// main statemachine of base controller
CASE me.StateMachine.intState OF
    cSTA_PONBusy: 
        THIS^.sta_PONBusy();
    cSTA_PON: 
        THIS^.sta_PON();
	cSTA_OFFBusy: 
        THIS^.sta_OFFBusy();
    cSTA_OFF: 
        THIS^.sta_OFF();
    cSTA_ERROR: 
        THIS^.sta_ERROR();
    cSTA_ERRORQuit: 
        THIS^.sta_ERRORQuit();
	cSTA_EOFFBusy:
		THIS^.sta_EOFFBusy();
	cSTA_EOFF:
		THIS^.sta_EOFF();
    cSTA_SINGLE_ANSWER: 
        THIS^.sta_SINGLE_ANSWER();
END_CASE;
END_METHOD

END_FUNCTION_BLOCK

// POUs/BaseCtrl/I_CtrlBase
INTERFACE I_CtrlBase

PROPERTY CtrlCIf : POINTER TO T_Ctrl_CIf
GET
END_GET
END_PROPERTY

PROPERTY CtrlFB : POINTER TO FB_CtrlBASE
GET
END_GET
END_PROPERTY

END_INTERFACE

// POUs/Utility/Logger/BasLog/FB_BasLog
FUNCTION_BLOCK FB_BasLog
VAR_INPUT
END_VAR
VAR_OUTPUT
END_VAR
VAR
	stBlClientInfo : T_Bl_LibClient;
	stBlBaseStruct : T_Bl_BaseStruc;
	fbQueue : FB_Queue;
END_VAR

(*__________________________________________________________________________________________________
¦	
¦	Vistaprint Schweiz GmbH
¦	CH - 8401 Winterthur
¦
¦	www.vistaprint.ch - info@vistaprint.ch
¦___________________________________________________________________________________________________

Function desription:
Base logger system. The FUB must be called defined globally one time in PLC-program. After that the implemented 
sender and receiver must interact over the public methodes of the FB_BasLog.

History:
Version		Date			Author		Comment
---------------------------------------------------------------------------------------------------
0.00.1		14.07.2014		AVME/KVO	Start history
___________________________________________________________________________________________________*)

METHOD PUBLIC M_ChangeMask : UINT
VAR_INPUT
	In_strClientName: STRING(Queue.cMAX_NAME_LENGTH); // name of the client
	In_udiNewMask: UDINT;		// new filter mask which log type should be logged for this client
END_VAR
VAR
	usiCnt:USINT;
END_VAR
// change of filter mask
IF (stBlClientInfo.usiClientNr>0) THEN
	FOR usiCnt :=0 TO (stBlClientInfo.usiClientNr-1) BY 1 DO
		IF (In_strClientName=stBlClientInfo.stClient[usiCnt].strName) THEN
			stBlClientInfo.stClient[usiCnt].udiMask := In_udiNewMask;
			M_ChangeMask := 0;
			RETURN;
		END_IF
	END_FOR
END_IF
M_ChangeMask := BasLog.cERR_SYSTEM_NOT_FOUND;
END_METHOD

METHOD PROTECTED M_CheckValidLogType : BOOL
VAR_INPUT
	In_udiLogType : UDINT;
END_VAR
VAR
	ii : UINT;
	udiValue : UDINT := 1;
END_VAR
// check all 2er square
FOR ii :=1 TO 32 BY 1 DO
	// if result identic 
	IF (udiValue=In_udiLogType) THEN
		M_CheckValidLogType := TRUE;
		RETURN;
	END_IF
	udiValue := udiValue * 2; // if not ok multiply with 2
END_FOR
M_CheckValidLogType := FALSE;
END_METHOD

METHOD PUBLIC M_ClientInit : BOOL
VAR_INPUT
	In_strClientName: STRING(Queue.cMAX_NAME_LENGTH); // name of the client
	In_udiMask: UDINT;		// filter mask which log typ should be logged for this client
	In_uinNrOfElement: UINT;	// number of elements in queue
	In_p_fbTimeStamp: POINTER TO FB_TimeStamp; 
	In_bolUseLocalTimeStamp : BOOL; // use local time stamp or UTC
END_VAR
VAR_OUTPUT
	Out_pHandle: POINTER TO T_Queue_Info; 	// handle for read
	Out_uinStatus: UINT;	// feedback value 0:ok
END_VAR
VAR
	usiCnt: USINT;
	pQueueHandle : POINTER TO T_Queue_Info;
	pQueueSysHandle : POINTER TO T_Queue_SysInfo;
	uinStatus : UINT;
END_VAR

// client declaration
IF (stBlClientInfo.usiClientNr>0) THEN
	FOR usiCnt :=0 TO (stBlClientInfo.usiClientNr-1) BY 1 DO
		IF (In_strClientName=stBlClientInfo.stClient[usiCnt].strName) THEN
			// name allready exist - return handle
			Out_pHandle :=  ADR(stBlClientInfo.stHandleRow[0].pQueueHandle[usiCnt]);
			Out_uinStatus := 0;
			RETURN;
		END_IF
	END_FOR
END_IF

// entry timestamp FB
IF (In_p_fbTimeStamp=TC3_MEMMAN.NULL) THEN
	IF (stBlClientInfo.p_fbTimeStamp=TC3_MEMMAN.NULL) THEN
		Out_uinStatus := BasLog.cERR_NO_FB_TIME_STAMP_POINTER;
		RETURN;
	END_IF
ELSE
	stBlClientInfo.p_fbTimeStamp := In_p_fbTimeStamp;
END_IF

	
IF (stBlClientInfo.usiClientNr<BasLog.cMAX_CLIENTS) THEN
	// entry info of new client
	stBlClientInfo.stClient[stBlClientInfo.usiClientNr].strName := In_strClientName;
	stBlClientInfo.stClient[stBlClientInfo.usiClientNr].udiMask := In_udiMask;
	stBlClientInfo.stClient[stBlClientInfo.usiClientNr].udiNrOfElements := In_uinNrOfElement;
	stBlClientInfo.stClient[stBlClientInfo.usiClientNr].bolUseLocalTimeStamp := In_bolUseLocalTimeStamp;
		
	// init queue system if place for new client 
	fbQueue.M_Init(In_strQueueName:=In_strClientName,In_uinNrOfElement:=In_uinNrOfElement,In_udiSizeOfElement:=SIZEOF(T_Bl_BaseStruc),
					In_uinMode:=0,Out_pHandle=>pQueueSysHandle,Out_uinStatus=>uinStatus);
					
	// check feedback from init
	IF (uinStatus<>0) THEN
		Out_uinStatus := uinStatus; // error init queue system
	ELSE
		
		// return handle of TC field zero
		Out_pHandle := ADR(stBlClientInfo.stHandleRow[0].pQueueHandle[stBlClientInfo.usiClientNr]);
		
		// increment client count
		stBlClientInfo.usiClientNr := stBlClientInfo.usiClientNr + 1;
		
		// requirement for handles, if not allready done by tasks
		FOR usiCnt :=0 TO Queue.cMAX_NR_OF_TASKS BY 1 DO
			// if requests allready exist 
			IF (stBlClientInfo.stHandleRow[usiCnt].usiRequest<>0) THEN
				// check for handle
				uinStatus := fbQueue.M_GetHandle_TC(In_strQueueName:=In_strClientName,In_bytTaskIndex:=usiCnt, Out_pQueueHandle=>pQueueHandle);
				
				// check feedback from M_GetHandle_TC
				IF (uinStatus=0) AND (pQueueHandle<>TC3_MEMMAN.NULL) THEN
					// if no error entry handle
					stBlClientInfo.stHandleRow[usiCnt].pQueueHandle[stBlClientInfo.usiClientNr-1] := pQueueHandle;
					stBlClientInfo.stHandleRow[0].pQueueHandle[stBlClientInfo.usiClientNr-1] := pQueueHandle;
				ELSE
					Out_uinStatus := uinStatus; // error M_GetHandle_TC
				END_IF
 			END_IF
		END_FOR
	END_IF
					
ELSE
	Out_uinStatus := BasLog.cERR_TOO_MANY_CLIENTS;
	RETURN;
END_IF
END_METHOD

METHOD PUBLIC M_GetHandle : UINT
VAR_INPUT
;
END_VAR
VAR_OUTPUT
	Out_pHandle : POINTER TO T_Bl_LibHandleRow; // handle of log system for write (M_Log)
END_VAR
VAR
	fbGETCURTASKINDEX : GETCURTASKINDEX;
	usiCnt: USINT;
	pQueueHandle : POINTER TO BYTE;
	uinStatus : UINT;
END_VAR
// get handle of log system
fbGETCURTASKINDEX(); // This function block finds the task index of the task which is called from.
IF (stBlClientInfo.usiClientNr=0) THEN
	// set information that for this taskclass information are requested
	stBlClientInfo.stHandleRow[fbGETCURTASKINDEX.index].usiRequest := 1;
	Out_pHandle := ADR(stBlClientInfo.stHandleRow[fbGETCURTASKINDEX.index]);
ELSE
	// get handle for all declared clients
	FOR usiCnt :=0 TO (stBlClientInfo.usiClientNr-1) BY 1 DO
		M_GetHandle := fbQueue.M_GetHandle(In_strQueueName:=stBlClientInfo.stClient[usiCnt].strName,Out_pQueueHandle=>pQueueHandle);
		
		IF (M_GetHandle=0) AND (pQueueHandle<>TC3_MEMMAN.NULL) THEN
			stBlClientInfo.stHandleRow[fbGETCURTASKINDEX.index].usiRequest := 1;
			stBlClientInfo.stHandleRow[fbGETCURTASKINDEX.index].pQueueHandle[usiCnt] := pQueueHandle;
			
			// handle write in TC 0 writer for reading function
			stBlClientInfo.stHandleRow[0].pQueueHandle[usiCnt] := pQueueHandle;
		ELSE
			RETURN;
		END_IF
	END_FOR
	Out_pHandle := ADR(stBlClientInfo.stHandleRow[fbGETCURTASKINDEX.index]);
END_IF
END_METHOD

METHOD PUBLIC M_Log : UINT
VAR_INPUT
	In_pHandle : POINTER TO BYTE;
	In_udiLogType: UDINT; // log type
	In_intCtrlID: INT; // unique controllerID which has created this entry
	In_strText1: STRING(BasLog.cMAX_CHAR_TEXT1);	//information text1
	In_strText2: STRING(BasLog.cMAX_CHAR_TEXT2); // information text2
	In_dinPar1: DINT; // value parameter  1
	In_dinPar2: DINT; // value parameter  2
	In_dinPar3: DINT; // value parameter  3
	In_dinPar4: DINT; // value parameter  4
END_VAR
VAR
	stTimeStruct: TIMESTRUCT;
	pHandleRow: POINTER TO T_Bl_LibHandleRow;
	usiCnt:USINT;
	uinStatus:UINT;
END_VAR

// check handle ok
IF (In_pHandle=TC3_MEMMAN.NULL) THEN
	M_Log := BasLog.cERR_NO_HANDLE;
	RETURN;
END_IF

// check for correct logtyp
IF ((In_udiLogType>0) AND (M_CheckValidLogType(In_udiLogType)=TRUE))THEN
	// interprete input as row with handles
	pHandleRow := In_pHandle;
	// if time stamp fb is valid
	IF (stBlClientInfo.p_fbTimeStamp<>TC3_MEMMAN.NULL) THEN
		IF (stBlClientInfo.p_fbTimeStamp^.Out_bolInitOk=TRUE) THEN
			IF (stBlClientInfo.stClient[usiCnt].bolUseLocalTimeStamp=FALSE) THEN
				// write time in struct
				stTimeStruct :=  stBlClientInfo.p_fbTimeStamp^.UTC_TimeStruct;
			ELSE
				// write time in struct
				stTimeStruct := stBlClientInfo.p_fbTimeStamp^.LocalTime_TimeStruct_BaseWin;
			END_IF
		ELSE
			M_Log := BasLog.cERR_NO_FB_TIME_STAMP_INIT_NOT_OK;
			RETURN;
		END_IF
	ELSE
		M_Log := BasLog.cERR_NO_FB_TIME_STAMP_POINTER;
		RETURN;
	END_IF
	
	// write parameter and time in struct
	stBlBaseStruct.uinMs := stTimeStruct.wMilliseconds;
	stTimeStruct.wMilliseconds := 0; // The system time has a resolution of 1ms, while the resolution of DATE_AND_TIME is 1s. The milliseconds from the system time are used in the course of the conversion to determine the direction of rounding for the returned DATE_AND_TIME value. Set the wMilliseconds member of the Windows system time structure to zero to deactivate the rounding.
	stBlBaseStruct.dtDateTimeEntry := SYSTEMTIME_TO_DT(stTimeStruct);
	
	stBlBaseStruct.udiLogType := In_udiLogType;
	stBlBaseStruct.intCtrlID := In_intCtrlID;
	stBlBaseStruct.strText1 := In_strText1;
	stBlBaseStruct.strText2 := In_strText2;
	stBlBaseStruct.dinPar1 := In_dinPar1;
	stBlBaseStruct.dinPar2 := In_dinPar2;
	stBlBaseStruct.dinPar3 := In_dinPar3;
	stBlBaseStruct.dinPar4 := In_dinPar4;
	
	// send write command depending on filter mask
	IF (stBlClientInfo.usiClientNr>0) THEN
		FOR usiCnt :=0 TO (stBlClientInfo.usiClientNr-1) BY 1 DO
			// check filter mask
			IF ((In_udiLogType AND stBlClientInfo.stClient[usiCnt].udiMask)<>0) THEN
				uinStatus := fbQueue.M_Write(In_pQueueHandle:=pHandleRow^.pQueueHandle[usiCnt],In_pData:=ADR(stBlBaseStruct));
				IF (uinStatus<>0) THEN
					M_Log := uinStatus;
				END_IF
			END_IF
		END_FOR
	END_IF
ELSE
	M_Log := BasLog.cERR_INVALID_LOGTYPE;
END_IF
END_METHOD

METHOD PUBLIC M_Read : UINT
VAR_INPUT
	In_pHandle : POINTER TO POINTER TO BYTE; // handle for read
	In_pData: POINTER TO T_Bl_BaseStruc; // Pointer for feedback element
END_VAR
VAR
	pReadHandle : POINTER TO POINTER TO T_Queue_Info;
	usiCnt:USINT;
	uinStatus:UINT;
END_VAR

// check handle ok
IF (In_pHandle=TC3_MEMMAN.NULL) THEN
	M_Read := BasLog.cERR_NO_HANDLE;
	RETURN;
END_IF

IF (In_pHandle^=TC3_MEMMAN.NULL) THEN
	M_Read := BasLog.cERR_NO_WRITE_TASK;
	RETURN;
ELSE
	pReadHandle := In_pHandle;
	
	// readout
	M_Read := fbQueue.M_Read(In_pQueueHandle:= pReadHandle^,In_pData:=In_pData); // return<> -> error
END_IF
END_METHOD

END_FUNCTION_BLOCK

// POUs/Utility/Queue/FB_Queue
FUNCTION_BLOCK FB_Queue
VAR // buffer dynamic and PERSISTENT?????
	// creted with new -> dynamic but not retain....arrBuffer: ARRAY[0..ConstBaseLog.MAX_BUFFER_SIZE] OF BYTE; (* Buffer memory used by FB_MemRingBuffer function block *)
	stQueueLibInfo	: T_Queue_LibInfo;
END_VAR

(*__________________________________________________________________________________________________
¦	
¦	Vistaprint Schweiz GmbH
¦	CH - 8401 Winterthur
¦
¦	www.vistaprint.ch - info@vistaprint.ch
¦___________________________________________________________________________________________________

Function desription:
Queue functionallity for mutli tasking system. The FUB must be called defined globally one time in PLC-program. After that the implemented 
sender and receiver must interact over the public methodes.

Public methodes:

M_Clear: 
	Functionality: - Clear all queue entries
	Input parameter: - Queue handlings pointer In_pQueueHandle
	Methode return:	- Status UINT


History:
Version		Date			Author		Comment
---------------------------------------------------------------------------------------------------
0.00.1		14.07.2014		AVME/KVO	Start history
___________________________________________________________________________________________________*)

METHOD FB_exit : BOOL
VAR_INPUT
	bInCopyCode : BOOL; // if TRUE, the exit method is called for exiting an instance that is copied afterwards (online change).
END_VAR
VAR
	pSysInfo : POINTER TO T_Queue_SysInfo;
	pSysInfoNext : POINTER TO T_Queue_SysInfo;
	jj : USINT;
	usiCnt : USINT;
	pDelPointer : POINTER TO BYTE;
	pDelQueueInfo : POINTER TO T_Queue_Info;
END_VAR
END_METHOD

METHOD PROTECTED M_AllocNewQueue : POINTER TO BYTE

VAR_INPUT
	In_udiSizeOfQueue : UDINT; // Byte size of quee to allocate
END_VAR
// Debug counter
stQueueLibInfo.stSysDebugInfo.uinAllocnewQCalls := stQueueLibInfo.stSysDebugInfo.uinAllocnewQCalls + 1;
M_AllocNewQueue := __NEW(BYTE,In_udiSizeOfQueue);

// check if allocate memory is ok
IF (M_AllocNewQueue=TC3_MEMMAN.NULL) THEN
	stQueueLibInfo.uinFUBInternalError := Queue.cERR_MEM_ALLOC;
	M_AllocNewQueue := TC3_MEMMAN.NULL;
END_IF
END_METHOD

METHOD PROTECTED M_AllocNewQueueInfo : POINTER TO T_Queue_Info
VAR_INPUT
END_VAR
VAR
	pSysInfo : POINTER TO T_Queue_SysInfo;
END_VAR
// Debug counter
stQueueLibInfo.stSysDebugInfo.uinAllocNewQICalls := stQueueLibInfo.stSysDebugInfo.uinAllocNewQICalls + 1;

M_AllocNewQueueInfo := __NEW(T_Queue_Info);

// check if allocate memory is ok
IF (M_AllocNewQueueInfo=TC3_MEMMAN.NULL) THEN
	stQueueLibInfo.uinFUBInternalError := Queue.cERR_MEM_ALLOC;
	M_AllocNewQueueInfo := TC3_MEMMAN.NULL;
END_IF
END_METHOD

METHOD PROTECTED M_AllocNewQueueSystem : POINTER TO T_Queue_SysInfo
VAR_INPUT
END_VAR
VAR
	pSysInfo : POINTER TO T_Queue_SysInfo;
END_VAR
// Debug counter
stQueueLibInfo.stSysDebugInfo.uinAllocNewQSCalls := stQueueLibInfo.stSysDebugInfo.uinAllocNewQSCalls + 1;

M_AllocNewQueueSystem := __NEW(T_Queue_SysInfo);

// check if allocate memory is ok
IF (M_AllocNewQueueSystem=TC3_MEMMAN.NULL) THEN
	stQueueLibInfo.uinFUBInternalError := Queue.cERR_MEM_ALLOC;
	M_AllocNewQueueSystem := TC3_MEMMAN.NULL;
END_IF
END_METHOD

METHOD PROTECTED M_CheckAndAppendQueueSysInfo : POINTER TO T_Queue_SysInfo
VAR_INPUT
	In_strQueue : STRING(Queue.cMAX_NAME_LENGTH);
	In_bolCheckOnly : BOOL; // create not automaticallyy a new system -> feedback only valid if exist
END_VAR
VAR
	pSysInfo : POINTER TO T_Queue_SysInfo;
END_VAR
// methode check if queue system allready exist. If not allocate a new one and return pointer.
// Debug counter
stQueueLibInfo.stSysDebugInfo.uinCheckAndAppendQSCalls := stQueueLibInfo.stSysDebugInfo.uinCheckAndAppendQSCalls + 1;

// exist no queue system?
IF (stQueueLibInfo.pstQueue_SysInfo=TC3_MEMMAN.NULL) THEN
	// no queue system exist -> return
	IF (In_bolCheckOnly=TRUE) THEN
		M_CheckAndAppendQueueSysInfo := TC3_MEMMAN.NULL;
		RETURN;
	END_IF
	
	// allocate new queue system
	stQueueLibInfo.pstQueue_SysInfo := M_AllocNewQueueSystem();
	IF (stQueueLibInfo.pstQueue_SysInfo<>TC3_MEMMAN.NULL) THEN
		pSysInfo := stQueueLibInfo.pstQueue_SysInfo;
		// entry queue name
		pSysInfo^.strQueueName := In_strQueue;
		// add secure element
		pSysInfo^.udiSecure := Queue.cSECURE_CODE;
	
		M_CheckAndAppendQueueSysInfo := pSysInfo;
		RETURN;
	ELSE
		M_CheckAndAppendQueueSysInfo := TC3_MEMMAN.NULL;
		RETURN;
	END_IF
END_IF

IF (stQueueLibInfo.pstQueue_SysInfo<>TC3_MEMMAN.NULL) THEN
	// queue system allready exisit
	pSysInfo := stQueueLibInfo.pstQueue_SysInfo;
	
	WHILE (pSysInfo<>TC3_MEMMAN.NULL) DO
		// check queue name
		IF (pSysInfo^.strQueueName = In_strQueue) THEN
			// name found
			M_CheckAndAppendQueueSysInfo := pSysInfo;
			RETURN;
		END_IF
		
		// is this the last element?
		IF (pSysInfo^.pstNextQueue_SysInfo=TC3_MEMMAN.NULL) THEN
			// no queue system exist -> return
			IF (In_bolCheckOnly) THEN
				M_CheckAndAppendQueueSysInfo := TC3_MEMMAN.NULL;
				RETURN;
			END_IF
			
			// allocate new queue system
			pSysInfo^.pstNextQueue_SysInfo := M_AllocNewQueueSystem();
			
			IF (pSysInfo^.pstNextQueue_SysInfo<>TC3_MEMMAN.NULL) THEN
				// reference to new allocated queue system
				pSysInfo := pSysInfo^.pstNextQueue_SysInfo;
				// entry queue name
				pSysInfo^.strQueueName := In_strQueue;
				// add secure element
				pSysInfo^.udiSecure := Queue.cSECURE_CODE;
			
				M_CheckAndAppendQueueSysInfo := pSysInfo;
				RETURN;
			ELSE
				M_CheckAndAppendQueueSysInfo := TC3_MEMMAN.NULL;
				RETURN;
			END_IF
		END_IF
		
		// reference to next element
		pSysInfo := pSysInfo^.pstNextQueue_SysInfo;
	END_WHILE
END_IF

M_CheckAndAppendQueueSysInfo := TC3_MEMMAN.NULL;
END_METHOD

METHOD PUBLIC M_Clear : UINT
VAR_INPUT
	In_pQueueHandle : POINTER TO BYTE; // handle from M_GetHandle()
END_VAR
VAR
	pSysInfo : POINTER TO T_Queue_SysInfo;
	pInfo : POINTER TO T_Queue_Info;
	usiCnt: USINT;
END_VAR
// Clear specific queue system

// check handle ok
IF (In_pQueueHandle=TC3_MEMMAN.NULL) THEN
	M_Clear := Queue.cERR_HANDLE_INVALID;
	RETURN;
END_IF

// handle is pointer to queue info system
pInfo := In_pQueueHandle;

// for reading needed access to system info (check all task class queues)
IF (pInfo^.pQueueSysInfo=TC3_MEMMAN.NULL) THEN
	M_Clear := Queue.cERR_HANDLE_INVALID;
	RETURN;
END_IF

// access system info struct
pSysInfo := pInfo^.pQueueSysInfo;

// validate pointer
IF (pSysInfo^.udiSecure<>Queue.cSECURE_CODE) THEN
	M_Clear := Queue.cERR_HANDLE_INVALID;
	RETURN;
END_IF


// check all queues for first entry
// loop over all queues
FOR usiCnt :=0 TO Queue.cMAX_NR_OF_TASKS BY 1 DO
	pInfo := pSysInfo^.pQueueInfo[usiCnt];
	IF (pInfo<>TC3_MEMMAN.NULL) THEN
		IF (pInfo^.fbBuffer.pBuffer<>TC3_MEMMAN.NULL) THEN
			
			MEMSET( ADR( pInfo^.fbBuffer.pBuffer), 0, pInfo^.fbBuffer.cbBuffer); (* reset (optional) internal buffer *)
			pInfo^.fbBuffer.A_Reset( );
			
			IF (pInfo^.fbBuffer.bOk=TRUE) THEN
				pInfo^.udiFillLevel := (pInfo^.fbBuffer.cbSize * 100) / pInfo^.fbBuffer.cbBuffer; // % 0 empty queue
			ELSE
				M_Clear := Queue.cERR_CLEAR;
				RETURN;
			END_IF
		ELSE
			M_Clear := Queue.cERR_QUEUE_DOES_NOT_EXIST;
			RETURN;
		END_IF
	END_IF
END_FOR
END_METHOD

METHOD PUBLIC M_GetHandle : UINT
VAR_INPUT
	In_strQueueName: STRING(Queue.cMAX_NAME_LENGTH); // name of the queue system
END_VAR
VAR_OUTPUT
	Out_pQueueHandle : POINTER TO T_Queue_Info;
END_VAR
VAR
	fbGETCURTASKINDEX : GETCURTASKINDEX;
END_VAR
// get handle of a specific queue identification over name and task index
fbGETCURTASKINDEX(); // This function block finds the task index of the task which is called from.

// get handle based on task index
M_GetHandle := M_GetHandle_TC(In_strQueueName,fbGETCURTASKINDEX.index,Out_pQueueHandle=>Out_pQueueHandle);
END_METHOD

METHOD PUBLIC M_GetHandle_TC : UINT
VAR_INPUT
	In_strQueueName: STRING(Queue.cMAX_NAME_LENGTH); // name of the queue system
	In_bytTaskIndex: BYTE; // calling task index
END_VAR
VAR_Output
	Out_pQueueHandle : POINTER TO T_Queue_Info;
END_VAR
VAR
	pSysInfo : POINTER TO T_Queue_SysInfo;
	pInfo : POINTER TO T_Queue_Info;
	udiSizeOfQueue: UDINT;
END_VAR
// get handle of a specific queue identification over name and task index

// Debug counter
stQueueLibInfo.stSysDebugInfo.uinGetHandleCalls := stQueueLibInfo.stSysDebugInfo.uinGetHandleCalls + 1;

IF (In_strQueueName='') THEN
	M_GetHandle_TC := Queue.cERR_QUEUE_NAME;
	RETURN;
END_IF
IF (LEN(In_strQueueName)=0) THEN
	M_GetHandle_TC := Queue.cERR_QUEUE_NAME;
	RETURN;
END_IF

// check if queue system allready exist
pSysInfo := M_CheckAndAppendQueueSysInfo(In_strQueueName,FALSE); // false means check if queue system exist!!!

IF (pSysInfo=TC3_MEMMAN.NULL) THEN // system exist?
	M_GetHandle_TC := Queue.cERR_MEM_ALLOC;
	RETURN;
END_IF

// Queue exist and ready?
IF (pSysInfo^.pQueueInfo[In_bytTaskIndex-1]<>TC3_MEMMAN.NULL) THEN
	Out_pQueueHandle := pSysInfo^.pQueueInfo[In_bytTaskIndex-1];
	M_GetHandle_TC := 0;
ELSE
	pSysInfo^.pQueueInfo[In_bytTaskIndex-1] := M_AllocNewQueueInfo();
	
	IF (pSysInfo^.pQueueInfo[In_bytTaskIndex-1] <> TC3_MEMMAN.NULL) THEN
		pInfo := pSysInfo^.pQueueInfo[In_bytTaskIndex-1];
		pInfo^.pQueueSysInfo := pSysInfo; // save system info as reference in queue (parent)
		Out_pQueueHandle := pSysInfo^.pQueueInfo[In_bytTaskIndex-1];	//set pointer feedback
		
		// check if init/size definition allready done
		udiSizeOfQueue := UINT_TO_UDINT(pSysInfo^.uinNbrOfElement)*pSysInfo^.udiSizeOfElement;
		IF (udiSizeOfQueue<>0) THEN
			// Create queue and put reference to info structure
			pInfo^.fbBuffer.pBuffer := M_AllocNewQueue(udiSizeOfQueue);
			IF (pInfo^.fbBuffer.pBuffer<>TC3_MEMMAN.NULL) THEN
				//valid buffer allocated
				pInfo^.fbBuffer.cbBuffer := udiSizeOfQueue; // size created in byte
			ELSE
				M_GetHandle_TC := Queue.cERR_MEM_ALLOC;
				RETURN;
			END_IF
		ELSE
			pInfo^.bolAllocMe := TRUE; // get handle called before valid init done!
		END_IF
	ELSE
		M_GetHandle_TC := Queue.cERR_MEM_ALLOC;
		RETURN;
	END_IF
END_IF
END_METHOD

METHOD PUBLIC M_Init : BOOL
VAR_INPUT
	In_strQueueName: STRING(Queue.cMAX_NAME_LENGTH); // name of the queue system
	In_uinNrOfElement: UINT;		// number of queue element
	In_udiSizeOfElement: UDINT;	// size of an element
	In_uinMode:UINT;				// 0: no overwrite of buffer, 1: ring buffer overwrite oldest entry
END_VAR
VAR_OUTPUT
	Out_pHandle: POINTER TO T_Queue_SysInfo; 			// handle for every task class sender/receiver
	Out_uinStatus: UINT;			// error -> 0:ok
END_VAR
VAR
	pSysInfo : POINTER TO T_Queue_SysInfo;
	pInfo : POINTER TO T_Queue_Info;
	usiCnt: USINT;
	pByte : POINTER TO BYTE;
END_VAR
// Debug counter
stQueueLibInfo.stSysDebugInfo.uinIniCalls := stQueueLibInfo.stSysDebugInfo.uinIniCalls + 1;

IF (In_strQueueName='') THEN
	Out_uinStatus := Queue.cERR_QUEUE_NAME;
	RETURN;
END_IF
IF (LEN(In_strQueueName)=0) THEN
	Out_uinStatus := Queue.cERR_QUEUE_NAME;
	RETURN;
END_IF
IF (In_uinNrOfElement=0) THEN
	Out_uinStatus := Queue.cERR_NR_OF_ELEMENTS;
	RETURN;
END_IF
IF (In_udiSizeOfElement=0) THEN
	Out_uinStatus := Queue.cERR_SIZE_OF_ELEMENTS;
	RETURN;
END_IF

// check if queue system allready exist
pSysInfo := M_CheckAndAppendQueueSysInfo(In_strQueueName,FALSE); // false means check and if not exist create new queeue system!!!

IF (pSysInfo=TC3_MEMMAN.NULL) THEN // system exist
	Out_uinStatus := Queue.cERR_MEM_ALLOC;
	RETURN;
END_IF

// save buffer dimension
pSysInfo^.uinNbrOfElement := In_uinNrOfElement;
pSysInfo^.udiSizeOfElement := In_udiSizeOfElement;
pSysInfo^.uinMode := In_uinMode;

FOR usiCnt :=0 TO Queue.cMAX_NR_OF_TASKS BY 1 DO
	pInfo := pSysInfo^.pQueueInfo[usiCnt]; // Queue info allready allocated -> allocate missing queues for the queue info (init after get_handle)
	IF (pInfo<>TC3_MEMMAN.NULL) THEN // Queue Info allready exist?
		// queue allready allocated?
		IF (pInfo^.fbBuffer.pBuffer=TC3_MEMMAN.NULL) AND (pInfo^.bolAllocMe=TRUE) THEN
			// not allready allocated
			// create FIFO System
			pInfo^.fbBuffer.pBuffer := M_AllocNewQueue(UDINT_TO_UINT(In_uinNrOfElement*In_udiSizeOfElement));
			IF (pInfo^.fbBuffer.pBuffer<>TC3_MEMMAN.NULL) THEN
				//valid buffer allocated
				pInfo^.fbBuffer.cbBuffer := UINT_TO_UDINT(In_uinNrOfElement)*In_udiSizeOfElement; // size created in byte
				pInfo^.bolAllocMe := FALSE;	
			END_IF
		END_IF
	END_IF
END_FOR

Out_uinStatus := 0;
Out_pHandle := pSysInfo;
RETURN;
END_METHOD

METHOD PUBLIC M_Read : UINT
VAR_INPUT
	In_pQueueHandle : POINTER TO BYTE; // handle from M_GetHandle()
	In_pData: POINTER TO BYTE; // destination address of the read element
END_VAR
VAR
	pSysInfo : POINTER TO T_Queue_SysInfo;
	pInfo : POINTER TO T_Queue_Info;
	usiCnt: USINT;
END_VAR
// Reset specific queue system

// check handle ok
IF (In_pQueueHandle=TC3_MEMMAN.NULL) THEN
	M_Read := Queue.cERR_HANDLE_INVALID;
	RETURN;
END_IF

// handle is pointer to queue info system
pInfo := In_pQueueHandle;

// for reading needed access to system info (check all task class queues)
IF (pInfo^.pQueueSysInfo=TC3_MEMMAN.NULL) THEN
	M_Read := Queue.cERR_HANDLE_INVALID;
	RETURN;
END_IF

// access system info struct
pSysInfo := pInfo^.pQueueSysInfo;

// validate pointer
IF (pSysInfo^.udiSecure<>Queue.cSECURE_CODE) THEN
	M_Read := Queue.cERR_HANDLE_INVALID;
	RETURN;
END_IF

//check data read pointer
IF (In_pData=TC3_MEMMAN.NULL) THEN
	M_Read := Queue.cERR_DATA_INVALID;
	RETURN;
END_IF

// check all queues for first entry
// loop over all queues
FOR usiCnt :=0 TO Queue.cMAX_NR_OF_TASKS BY 1 DO
	pInfo := pSysInfo^.pQueueInfo[usiCnt];
	IF (pInfo<>TC3_MEMMAN.NULL) THEN
		
		IF (pInfo^.fbBuffer.pBuffer<>TC3_MEMMAN.NULL) THEN
			
			IF (pInfo^.fbBuffer.nCount>0) THEN // entry?
				pInfo^.fbBuffer.A_RemoveHead(pRead:= In_pData, cbRead:= pSysInfo^.udiSizeOfElement);

				pInfo^.udiFillLevel := (pInfo^.fbBuffer.cbSize * 100) / pInfo^.fbBuffer.cbBuffer;;
				M_Read := 0;
				RETURN;
			END_IF
		ELSE
			M_Read := Queue.cERR_QUEUE_DOES_NOT_EXIST;
			RETURN;
		END_IF
	END_IF
END_FOR

// queue empty
M_Read := Queue.cERR_QUEUE_EMPTY;
END_METHOD

METHOD PUBLIC M_ReadReference : UINT
VAR_INPUT
	In_pQueueHandle : POINTER TO BYTE; // handle from M_GetHandle()
END_VAR
VAR_OUTPUT
	Out_pData: POINTER TO BYTE; // read reference
END_VAR
VAR
	pSysInfo : POINTER TO T_Queue_SysInfo;
	pInfo : POINTER TO T_Queue_Info;
	usiCnt: USINT;
END_VAR
// get reference to element from queue 

// check handle ok
IF (In_pQueueHandle=TC3_MEMMAN.NULL) THEN
	M_ReadReference := Queue.cERR_HANDLE_INVALID;
	RETURN;
END_IF

// handle is pointer to queue info system
pInfo := In_pQueueHandle;

// for reading needed access to system info (check all task class queues)
IF (pInfo^.pQueueSysInfo=TC3_MEMMAN.NULL) THEN
	M_ReadReference := Queue.cERR_HANDLE_INVALID;
	RETURN;
END_IF

// access system info struct
pSysInfo := pInfo^.pQueueSysInfo;

// validate pointer
IF (pSysInfo^.udiSecure<>Queue.cSECURE_CODE) THEN
	M_ReadReference := Queue.cERR_HANDLE_INVALID;
	RETURN;
END_IF

// check all queues for first entry
// loop over all queues
FOR usiCnt :=0 TO Queue.cMAX_NR_OF_TASKS BY 1 DO
	pInfo := pSysInfo^.pQueueInfo[usiCnt];
	IF (pInfo<>TC3_MEMMAN.NULL) THEN
		IF (pInfo^.fbBuffer.pBuffer<>TC3_MEMMAN.NULL) THEN
			
			IF (pInfo^.fbBuffer.nCount>0) THEN // entry?
				pInfo^.fbBuffer.A_GetHead( 	pRead:= Out_pData, cbRead:= pSysInfo^.udiSizeOfElement);
				M_ReadReference := 0;
				RETURN;
			END_IF
		ELSE
			M_ReadReference := Queue.cERR_QUEUE_DOES_NOT_EXIST;
			RETURN;
		END_IF
	END_IF
END_FOR

// queue empty
M_ReadReference := Queue.cERR_QUEUE_EMPTY;
END_METHOD

METHOD PUBLIC M_Write : UINT
VAR_INPUT
	In_pQueueHandle : POINTER TO T_Queue_Info; // handle from M_GetHandle()
	In_pData: POINTER TO BYTE;  // source address of the write element
END_VAR
VAR
	pSysInfo : POINTER TO T_Queue_SysInfo;
	pInfo : POINTER TO T_Queue_Info;
	pData : POINTER TO BYTE; // read dummy element for remove oldest...
END_VAR
// Write element to specific queue system

// check handle ok
IF (In_pQueueHandle=TC3_MEMMAN.NULL) THEN
	M_Write := Queue.cERR_HANDLE_INVALID;
	RETURN;
END_IF

// handle is pointer to queue info system
pInfo := In_pQueueHandle;

// for reading needed access to system info (check all task class queues)
IF (pInfo^.pQueueSysInfo=TC3_MEMMAN.NULL) THEN
	M_Write := Queue.cERR_HANDLE_INVALID;
	RETURN;
END_IF

// access system info struct
pSysInfo := pInfo^.pQueueSysInfo;

// validate pointer
IF (pSysInfo^.udiSecure<>Queue.cSECURE_CODE) THEN
	M_Write := Queue.cERR_HANDLE_INVALID;
	RETURN;
END_IF

//check data
IF (In_pData=TC3_MEMMAN.NULL) THEN
	M_Write := Queue.cERR_DATA_INVALID;
	RETURN;
END_IF

// check if queue exist
IF (pInfo^.fbBuffer.pBuffer=TC3_MEMMAN.NULL) THEN
	M_Write := Queue.cERR_QUEUE_DOES_NOT_EXIST;
	RETURN;
END_IF


// check fill level
// feedback of FIFO = false -> overflow .... IF (pInfo^.udiFillLevel<100) AND (pInfo^.fbBuffer.nCount<pSysInfo^.uinNbrOfElement)THEN
pInfo^.fbBuffer.A_AddTail( pWrite:= In_pData,
				cbWrite:= pSysInfo^.udiSizeOfElement); 
(*				pBuffer:= ADR( arrBuffer ),
				cbBuffer:= SIZEOF( arrBuffer ),
				bOk=> Out_bolOk,
				nCount => Out_udiCount*)
IF (pInfo^.fbBuffer.bOk=FALSE) THEN (* overflow ? *)
	IF (pSysInfo^.uinMode=0) THEN //0:FIFO ring buffer overwrite
		IF (pData = TC3_MEMMAN.NULL) THEN // alloc new dummy read element
			pData := __NEW(BYTE,pSysInfo^.udiSizeOfElement);
		END_IF
		IF (pData <> TC3_MEMMAN.NULL) THEN // alloc new dummy read element
			pInfo^.fbBuffer.A_RemoveHead(pRead:= pData, cbRead:= pSysInfo^.udiSizeOfElement); (* remove one oldest entry *)
			__DELETE(pData); // release dummy memory
			
			pInfo^.fbBuffer.A_AddTail();
			pInfo^.udiFillLevel := (pInfo^.fbBuffer.cbSize * 100) / pInfo^.fbBuffer.cbBuffer;
			M_Write :=0; //Done
		ELSE
			M_Write := Queue.cERR_QUEUE_FULL;
		END_IF
		RETURN;
	ELSE
		pInfo^.udiFillLevel := (pInfo^.fbBuffer.cbSize * 100) / pInfo^.fbBuffer.cbBuffer;
		M_Write := Queue.cERR_QUEUE_FULL;
		RETURN;
	END_IF
ELSE
	pInfo^.udiFillLevel := (pInfo^.fbBuffer.cbSize * 100) / pInfo^.fbBuffer.cbBuffer;
	M_Write :=0; //Done
	RETURN;
END_IF
END_METHOD

END_FUNCTION_BLOCK

// POUs/Utility/getStrInstanceName
FUNCTION getStrInstanceName : T_MaxString
VAR_INPUT
	///'C:\TwinCAT\Plc\Project01\Data.txt';
	strPathName: T_MaxString;
END_VAR
VAR
	strDrive: STRING(3);
	strDir: T_MaxString;
	strFileName: T_MaxString;
	strExt: T_MaxString;
	bolSuccess: BOOL;
END_VAR


bolSuccess := F_SplitPathName( sPathName := strPathName,
                                sDrive := strDrive,
                                sDir := strDir,
                                sFileName := strFileName,
                                sExt := strExt );
								
								getStrInstanceName := MID (strExt,TC2_STANDARD.LEN(strExt),2);

END_FUNCTION

// POUs/Utility/DLL (Double Linked List)/FB_DLL
FUNCTION_BLOCK FB_DLL
VAR
	bDoDataWipe: BOOL := FALSE;
	pFirstElement: POINTER TO T_Element;
	pLastElement: POINTER TO T_Element;
	uiNumberOfElements: UINT;
END_VAR

METHOD addElement : POINTER TO T_Element
VAR_INPUT
	In_pData: POINTER TO BYTE;
	In_uliKey: ULINT;
END_VAR
VAR
	pCurrentElement: POINTER TO T_Element;
END_VAR
addElement := TC3_MEMMAN.NULL;

IF (pFirstElement = TC3_MEMMAN.NULL) THEN
	pCurrentElement := __NEW(T_Element);
	pFirstElement := pCurrentElement;
	pLastElement := pCurrentElement;
	pCurrentElement^.pPrevElement := TC3_MEMMAN.NULL;
	pCurrentElement^.pNextElement := TC3_MEMMAN.NULL;
	pCurrentElement^.pData := In_pData;
	pCurrentElement^.uliKey := In_uliKey;
	addElement := pCurrentElement;
ELSE
	pCurrentElement := __NEW(T_Element);
	pCurrentElement^.pPrevElement := pLastElement;
	pCurrentElement^.pNextElement := TC3_MEMMAN.NULL;
	pCurrentElement^.pData := In_pData;
	pCurrentElement^.uliKey := In_uliKey;
	pLastElement^.pNextElement := pCurrentElement;
	pLastElement := pCurrentElement;
	addElement := pCurrentElement;
END_IF

uiNumberOfElements := uiNumberOfElements + 1;
END_METHOD

METHOD deleteAll : POINTER TO T_Element
WHILE (pFirstElement <> TC3_MEMMAN.NULL) DO
	__DELETE(pFirstElement^.pData);
	deleteElement(pFirstElement);
END_WHILE
END_METHOD

METHOD deleteElement : POINTER TO BYTE
VAR_INPUT
	In_pDeleteElement: POINTER TO T_Element;
END_VAR
deleteElement := In_pDeleteElement^.pData;

IF bDoDataWipe THEN
	IF (In_pDeleteElement^.pData <> TC3_MEMMAN.NULL) THEN
		__DELETE(In_pDeleteElement^.pData);
	END_IF
	deleteElement := TC3_MEMMAN.NULL;
END_IF

IF (In_pDeleteElement = pFirstElement AND In_pDeleteElement = pLastElement) THEN
	pFirstElement := TC3_MEMMAN.NULL;
	pLastElement := TC3_MEMMAN.NULL;
ELSIF (In_pDeleteElement = pFirstElement) THEN
	pFirstElement := In_pDeleteElement^.pNextElement;
	In_pDeleteElement^.pNextElement^.pPrevElement := TC3_MEMMAN.NULL;
ELSIF (In_pDeleteElement = pLastElement) THEN
	pLastElement := In_pDeleteElement^.pPrevElement;
	In_pDeleteElement^.pPrevElement^.pNextElement := TC3_MEMMAN.NULL;
ELSE
	In_pDeleteElement^.pPrevElement^.pNextElement := In_pDeleteElement^.pNextElement;
	In_pDeleteElement^.pNextElement^.pPrevElement := In_pDeleteElement^.pPrevElement;
END_IF

__DELETE(In_pDeleteElement);

uiNumberOfElements := uiNumberOfElements - 1;
END_METHOD

METHOD FB_init : BOOL
VAR_INPUT
	/// if TRUE, the retain variables are initialized (warm start / cold start)
	bInitRetains: BOOL;
	/// if TRUE, the instance afterwards gets moved into the copy code (online change)
	bInCopyCode: BOOL;
	/// if TRUE, the stored data object are automatically deleted
	In_bDoDataWipe: BOOL;
END_VAR
pFirstElement := TC3_MEMMAN.NULL;
pLastElement := TC3_MEMMAN.NULL;
uiNumberOfElements := 0;

bDoDataWipe := In_bDoDataWipe;
END_METHOD

METHOD firstElement : POINTER TO T_Element
firstElement := pFirstElement;
END_METHOD

METHOD numberOfElements : UINT
numberOfElements := uiNumberOfElements;
END_METHOD

METHOD searchElement : POINTER TO T_Element
VAR_INPUT
	In_uliKey: ULINT;
END_VAR
VAR
	pCurrentElement: POINTER TO T_Element;
END_VAR
searchElement := TC3_MEMMAN.NULL;
pCurrentElement := pFirstElement;

WHILE (pCurrentElement <> TC3_MEMMAN.NULL) DO
	IF (pCurrentElement^.uliKey = In_uliKey) THEN
		searchElement := pCurrentElement;
		EXIT;
	END_IF
	pCurrentElement := pCurrentElement^.pNextElement;
END_WHILE
END_METHOD

END_FUNCTION_BLOCK

// POUs/Utility/FileFolder/FB_FileCopy
FUNCTION_BLOCK PUBLIC FB_FileCopy
VAR_INPUT
        srcNetId        : T_AmsNetId;   (* TwinCAT network address of the source file *)
        srcFileName     : T_MaxString;  (* source file path and name *)
        destNetId       : T_AmsNetId;   (* TwinCAT network address of the destination file *)
        destFileName    : T_MaxString;          (* destination file path and name *)
        bExecute        : BOOL;         (* rising edge starts fb execution *)
        tAdsTimeOut     : TIME;         (* ads timeout *)
END_VAR
VAR_OUTPUT
        bBusy           :BOOL;
        bError          :BOOL;
        nErrId          :UDINT;
END_VAR
VAR
        fbFileOpen      :FB_FileOpen;
        fbFileClose     :FB_FileClose;
        fbFileRead      :FB_FileRead;
        fbFileWrite     :FB_FileWrite;

        hSrcFile                :UINT   := 0;(* file handle of the source file *)
        hDestFile               :UINT   := 0;(* file handle of the destination file *)

        Step            :DWORD;
        RisingEdge      :R_TRIG;

        buffRead        :ARRAY[1..10000] OF BYTE;(* buffer *)
        cbReadLength    :UDINT:=0;
END_VAR

(*__________________________________________________________________________________________________
¦	
¦	Vistaprint Schweiz GmbH
¦	CH - 8401 Winterthur
¦
¦	www.vistaprint.ch - info@vistaprint.ch
¦___________________________________________________________________________________________________

Function desription:
	Copy functionality 
	!!!!!!direct source copy from example from Beckhoff -> not Vistaprint notation!!!!
		
History:
Version		Date			Author		Comment
---------------------------------------------------------------------------------------------------
0.00.1		14.05.2014		AVME/KVO	Start history
___________________________________________________________________________________________________*)



RisingEdge(CLK:=bExecute);
IF RisingEdge.Q THEN
        IF NOT bBusy THEN
                bBusy := TRUE;
                bError:= FALSE;
                nErrId:=0;
                Step := 1;
                cbReadLength:=0;
                hSrcFile:=0;
                hDestFile:=0;
        END_IF
END_IF


CASE Step OF
        0:(* do nothing *)
        ;

        1:(* open source file *)
        fbFileOpen(  bExecute := FALSE  );
        fbFileOpen(     sNetId := srcNetId,
                sPathName := srcFileName,
                nMode := FOPEN_MODEREAD OR FOPEN_MODEBINARY,
                ePath := PATH_GENERIC,
                tTimeout := tAdsTimeout,
                bExecute := TRUE );
                Step := Step + 1;

        2:
        fbFileOpen( bExecute := FALSE );
        IF ( NOT fbFileOpen.bBusy ) THEN
                IF ( fbFileOpen.bError ) THEN
                        nErrId := fbFileOpen.nErrId;
                        bError := TRUE;
                        Step := 50;
                ELSE
                        hSrcFile := fbFileOpen.hFile;
                        Step := Step + 1;
                END_IF
        END_IF

        3:(* open destination file *)
        fbFileOpen(  bExecute := FALSE  );
        fbFileOpen(     sNetId := destNetId,
                        sPathName := destFileName,
                        nMode := FOPEN_MODEWRITE OR FOPEN_MODEBINARY,
                        ePath := PATH_GENERIC,
                        tTimeout := tAdsTimeout,
                        bExecute := TRUE );
        Step := Step+1;

        4:
        fbFileOpen(  bExecute := FALSE  );
        IF ( NOT fbFileOpen.bBusy ) THEN
                IF ( fbFileOpen.bError ) THEN
                        nErrId := fbFileOpen.nErrId;
                        bError := TRUE;
                        Step := 50;
                ELSE
                        hDestFile := fbFileOpen.hFile;
                        Step := Step + 1;
                END_IF
        END_IF

        5:(*read data from source file*)
        cbReadLength := 0;
        fbFileRead( bExecute:= FALSE );
        fbFileRead(     sNetId:=SrcNetId,
                        hFile:=hSrcFile,
                        pReadBuff:= ADR(buffRead),
                        cbReadLen:= SIZEOF(buffRead),
                        bExecute:=TRUE,
                        tTimeout:=tAdsTimeOut );
        Step := Step + 1;

        6:
        fbFileRead( bExecute:= FALSE );
        IF ( NOT fbFileRead.bBusy ) THEN
                IF ( fbFileRead.bError ) THEN
                        nErrId := fbFileRead.nErrId;
                        bError := TRUE;
                        Step := 50;
                ELSE
                        cbReadLength := fbFileRead.cbRead;
                        Step := Step + 1;
                END_IF
        END_IF

        7:(*write data to destination file*)
        fbFileWrite( bExecute := FALSE );
        fbFileWrite(    sNetId:=DestNetId,
                        hFile:=hDestFile,
                        pWriteBuff:= ADR(buffRead),
                        cbWriteLen:= cbReadLength,
                        bExecute:=TRUE,
                        tTimeout:=tAdsTimeOut );
        Step := Step + 1;

        8:
        fbFileWrite( bExecute := FALSE );
        IF ( NOT fbFileWrite.bBusy ) THEN
                IF ( fbFileWrite.bError ) THEN
                        nErrId := fbFileWrite.nErrId;
                        bError := TRUE;
                        Step := 50;
                ELSE
                        IF fbFileRead.bEOF THEN (*Check if the EOF flag ist set *)
                                Step := 50;(*cleanup: close the destination and source files *)
                        ELSE
                                Step := 5; (* repeat reading *)
                        END_IF
                END_IF
        END_IF

        30:(* close the destination file *)
        fbFileClose( bExecute := FALSE );
        fbFileClose(    sNetId:=destNetId,
                        hFile:=hDestFile,
                        bExecute:=TRUE,
                        tTimeout:=tAdsTimeOut );
        Step := Step + 1;

        31:
        fbFileClose( bExecute := FALSE );
        IF ( NOT fbFileClose.bBusy ) THEN
                IF ( fbFileClose.bError ) THEN
                        nErrId := fbFileClose.nErrId;
                        bError := TRUE;
                END_IF
                Step := 50;
                hDestFile := 0;
        END_IF

        40: (* close source file *)
        fbFileClose( bExecute := FALSE );
        fbFileClose(    sNetId:=srcNetId,
                        hFile:=hSrcFile,
                        bExecute:=TRUE,
                        tTimeout:=tAdsTimeOut );
        Step := Step + 1;

        41:
        fbFileClose( bExecute := FALSE );
        IF ( NOT fbFileClose.bBusy ) THEN
                IF ( fbFileClose.bError ) THEN
                        nErrId := fbFileClose.nErrId;
                        bError := TRUE;
                END_IF
                Step := 50;
                hSrcFile := 0;
        END_IF

        50: (*error or ready => cleanup*)
        IF ( hDestFile <> 0 ) THEN
                Step := 30; (* close the destination file*)
        ELSIF (hSrcFile <> 0 ) THEN
                Step := 40; (* close the source file *)
        ELSE
                Step := 0;      (* ready *)
                bBusy := FALSE;
        END_IF

END_CASE

END_FUNCTION_BLOCK

// POUs/Utility/FileFolder/FB_FileHdl
FUNCTION_BLOCK FB_FileHdl

VAR_OUTPUT
	Out_bolBusy : BOOL; // busy
	Out_bolNewFileCreated : BOOL; // new file created -> set until next job -> possibility to write header
	Out_udiErrId : UDINT; // error id
	Out_strInfo : STRING; //
END_VAR
VAR
	uinStep : UINT;
	uinStep_old : UINT;
	uinSubStep : UINT;
	intCmd : INT;
	bolInitDone : BOOL;
	strNetId : STRING(23);
	strPathName : T_MaxString; 	// Contains the path and filename for the file to be opened. Note: The path can only point to the local computer’s file system! This means that network paths can not be used here!
	strPath : T_MaxString; 	// Contains only the path 
	strFileName : T_MaxString;	// Contains only the filename
	strFileExt : T_MaxString;	// Contains only the ext
	strPathNameArchive : T_MaxString; // string name of last copied archive file
	strTemp : T_MaxString;
	strFileNameTemp : STRING(200);
	strFullFileName : T_MaxString;
	intLenTemp : INT;
	uin_FileHandle : UINT;	//Contains the file handle created for the file when opening has been successful.
	pWriteBuff: POINTER TO BYTE; // Write buffer adress
	udiWriteLen : UDINT; // Write buffer len
	lreCurFileSize : LREAL;
	stNewestFileEntry : ST_FindFileEntry;
	fbFileOpen_1 : FB_FileOpen;
	fbFileClose_1 : FB_FileClose;
	fbFileWrite_1 : FB_FileWrite;
	fbFileDelete_1 : FB_FileDelete;
	fbFileRename_1 : FB_FileRename;
	fbFileCopy_1 : FB_FileCopy;
	fbFolderHdl_1 : FB_FolderHdl;
	lreMaxFileSize : LREAL := 10; //Bytes? maximal allowed filesize for file -> archivate and deleter or create new
	bolNewFileCreated : BOOL;
	bolTimeRead : BOOL;
	strActualTime : T_MaxString;
	fbNT_GetTime : NT_GetTime;
END_VAR
VAR CONSTANT
	// specific steps definitions
	cStep_Start: UINT := 501;
	cStep_StartReadingFilesInFolder: UINT := 502;
	cStep_ReadingFileInFolder: UINT := 504;
	cStep_FileDelete: UINT := 100;
	cStep_FileClose: UINT := 101;
	cStep_FileOpen: UINT := 102;
	cStep_FileWrite: UINT := 103;
	cStep_NewFile: UINT := 104;
	cStep_FileArchive: UINT := 105;
	cStep_Wait4Job: UINT := 500;
	cStep_Error: UINT := 256;
	
	cSubStep_Done: UINT := 0;
	cSubStep_Finished: UINT := 100;
	cSubStep_Error: UINT := 256;
	
	// configuration constants
	usiMode : UINT := 1; // Mode = 0 logfiles with date, =1 logfile with archive and date
	strSufixArchive : T_MaxString := '_Archive_';

	// commandes constants
	cFILE_HDL_CMD_DONE : INT := -1;
	cFILE_HDL_CMD_WRITE : INT := 1;
	cFILE_HDL_CMD_NEW_FILE : INT := 2;
	cFILE_HDL_CMD_REFRESH_FILE_LIST : INT := 3;
	cFILE_HDL_CMD_CLOSE : INT := 4;
	cFILE_HDL_CMD_FILE_DELETE : INT := 5;
END_VAR

(*__________________________________________________________________________________________________
¦	
¦	Vistaprint Schweiz GmbH
¦	CH - 8401 Winterthur
¦
¦	www.vistaprint.ch - info@vistaprint.ch
¦___________________________________________________________________________________________________

Function desription:
	Manage folder with files: 
	Cyclic Actions:
		- todo evtl. in folder hdl... create folder
		- open file ("a+": Opens for reading and appending; the appending operation includes the removal of the EOF marker before new data is written to the file and the EOF marker is restored after writing is complete; creates the file first if it doesn’t exist.
					When a file is opened with the "a" or "a+" access type, all write operations occur at the end of the file. The file pointer can be repositioned using FB_FileSeek, but is always moved back to the end of the file before any write operation is carried out. Thus, existing data cannot be overwritten.)
		- add buffer to file
		- close file
		- delete file
		- archivate file
		- supervision of active file size
		- todo supervision of nr of entries
		
History:
Version		Date			Author		Comment
---------------------------------------------------------------------------------------------------
0.00.1		13.05.2014		AVME/KVO	Start history
___________________________________________________________________________________________________*)

// read out actual TIME
fbNT_GetTime.START := FALSE;
fbNT_GetTime();
fbNT_GetTime.NETID := '';
fbNT_GetTime.START := TRUE;
fbNT_GetTime.TMOUT := T#500MS;
fbNT_GetTime();

fbFolderHdl_1(); // cyclic call for supervision of numbers of file in folder

CASE uinStep OF
	0:	
		Out_strInfo := 'Wait for init ok -> call methode M_INIT()';
		Out_bolBusy := TRUE;
		IF (bolInitDone=TRUE) AND (fbFolderHdl_1.Out_bolInitDone=TRUE) THEN // refresh file list done
			uinStep := cStep_Start;
		END_IF
		
	cStep_Start: 
		Out_strInfo := 'Start';	
		// entry action
		IF (uinStep<>uinStep_old) THEN
			Out_bolBusy := TRUE;
			Out_udiErrId := 0;
			uinStep_old := uinStep;
			fbFolderHdl_1(); // -> set bol busy
		END_IF

		stNewestFileEntry := fbFolderHdl_1.get_NewestFileEntry; // automatic refresh list!!!
		
		IF ((stNewestFileEntry.sFileName<>'') AND (FIND(stNewestFileEntry.sFileName,strFileName)<>0) AND (FIND(stNewestFileEntry.sFileName,strFileExt)<>0)) THEN // not empty -> found entry and contains IN_strFileName -> no change in config
			IF (usiMode = 0) THEN //new file name with Date and time sufix
				(*???intLenTemp := LEN(stNewestFileEntry.sFileName)-FIND(stNewestFileEntry.sFileName,strFileExt)-1;
				strFileName := stNewestFileEntry.sFileName;
				strFileName := MID (strFileName, 1,intLenTemp); // LEFT doesn't work????
				strPathName := THIS^.M_GetPathName(In_bolSufixDateTime:=FALSE,In_strSufixBeforeDateTime:='');	*)
				strPathName := CONCAT(STR1:=strPath,STR2:=stNewestFileEntry.sFileName);
				lreCurFileSize := UINT64_TO_LREAL(stNewestFileEntry.fileSize); // size of existing file
			ELSE
				// new file name stay always the same -> get size
				strPathName := THIS^.M_GetPathName(In_bolSufixDateTime:=FALSE,In_strSufixBeforeDateTime:='');
				stNewestFileEntry := fbFolderHdl_1.M_getFileInfo(IN_strFileNameWithExt:=strPathName);
				lreCurFileSize := UINT64_TO_LREAL(stNewestFileEntry.fileSize); // size of existing file
			END_IF
			uinStep := cStep_Wait4Job;
		ELSE
			// no matching filename found -> create new file	
			IF (usiMode = 0) THEN // new file name with Date and time sufix
				strPathName := THIS^.M_GetPathName(In_bolSufixDateTime:=TRUE,In_strSufixBeforeDateTime:='_');	
			ELSE	// new file name stay the same but actual file archive with Date and time sufix
				
				strPathName := THIS^.M_GetPathName(In_bolSufixDateTime:=FALSE,In_strSufixBeforeDateTime:='');	
			END_IF
			lreCurFileSize := 0;
			uinStep := cStep_NewFile; // create a new file
		END_IF

	cStep_Wait4Job:	
		Out_strInfo := 'Wait for job';
		// entry action
		IF (uinStep<>uinStep_old) THEN
			Out_bolBusy := FALSE;
			uinSubStep := cSubStep_Done;
			uinStep_old := uinStep;
		END_IF
		
		
		IF (intCmd = cFILE_HDL_CMD_FILE_DELETE) THEN
			Out_bolBusy := TRUE;
			Out_bolNewFileCreated := FALSE;
			uinStep := cStep_FileDelete;
		END_IF
		
		IF (intCmd = cFILE_HDL_CMD_NEW_FILE) THEN
			Out_bolNewFileCreated := FALSE;
			Out_bolBusy := TRUE;
			IF ( uin_FileHandle <> 0 ) THEN // old file still open
				uinStep := cStep_FileClose;
			ELSE
				uinStep := cStep_NewFile;
			END_IF
		END_IF

		IF (intCmd = cFILE_HDL_CMD_WRITE) THEN
			Out_bolNewFileCreated := FALSE;
			Out_bolBusy := TRUE;
			IF ((lreCurFileSize + UDINT_TO_LREAL(udiWriteLen)) > lreMaxFileSize) THEN // supervision of filesize
				IF ( uin_FileHandle <> 0 ) THEN // no file open
					uinStep := cStep_FileClose;
				ELSE
					uinStep := cStep_NewFile;
				END_IF
			ELSE
				IF ( uin_FileHandle <> 0 ) THEN // no file open
					uinStep := cStep_FileWrite;
				ELSE
					uinStep := cStep_FileOpen;
				END_IF
			END_IF
		END_IF
		
		IF (intCmd = cFILE_HDL_CMD_CLOSE) THEN
			Out_bolNewFileCreated := FALSE;
			Out_bolBusy := TRUE;
			uinStep := cStep_FileClose;
		END_IF
		
	cStep_FileDelete:
		Out_strInfo := 'Delete file busy';	
		// entry action
		IF (uinStep<>uinStep_old) THEN
			Out_bolBusy := TRUE;
			uinSubStep := cSubStep_Done;
			uinStep_old := uinStep;
		END_IF
		
		THIS^.M_FileDelete(strNetId,strPathName);
		
		IF (uinSubStep = cSubStep_Finished) THEN
			IF (intCmd = cFILE_HDL_CMD_NEW_FILE) OR (intCmd = cFILE_HDL_CMD_WRITE) THEN
				uinStep := cStep_NewFile;
			ELSE
				uinStep := cStep_Wait4Job; 
			END_IF
		ELSIF (uinSubStep = cSubStep_Error) THEN
			intCmd := cFILE_HDL_CMD_DONE;
			uinStep := cStep_Error;
		END_IF
		
	cStep_NewFile:
		Out_strInfo := 'New file busy';
		// entry action
		IF (uinStep<>uinStep_old) THEN
			Out_bolBusy := TRUE;
			uinSubStep := cSubStep_Done;
			uinStep_old := uinStep;
		END_IF	
		
		lreCurFileSize := 0;
		
		IF (usiMode = 0) THEN // new file name with Date and time sufix
			strPathName := THIS^.M_GetPathName(In_bolSufixDateTime:=TRUE,In_strSufixBeforeDateTime:='');	
		ELSE
			// new file name stay the same but actual file archive with Date and time sufix
			strPathName := THIS^.M_GetPathName(In_bolSufixDateTime:=FALSE,In_strSufixBeforeDateTime:='');	
		END_IF
		
		bolNewFileCreated := TRUE;
		
		IF (intCmd = cFILE_HDL_CMD_WRITE) OR (intCmd = cFILE_HDL_CMD_NEW_FILE) THEN
			IF (usiMode = 0) THEN // new file name with Date and time sufix
				uinStep := cStep_FileOpen;
			ELSE
				uinStep := cStep_FileArchive;
			END_IF
		ELSE
			uinStep := cStep_FileOpen;
		END_IF	
	
	cStep_FileOpen:	
		Out_strInfo := 'Open file busy';
		// entry action
		IF (uinStep<>uinStep_old) THEN
			Out_bolBusy := TRUE;
			uinSubStep := cSubStep_Done;
			uinStep_old := uinStep;
		END_IF	

		THIS^.M_FileOpen(strNetId,strPathName);
		
		IF (uinSubStep = cSubStep_Finished) THEN
			IF (bolNewFileCreated) THEN
				Out_bolNewFileCreated := TRUE;
				bolNewFileCreated := FALSE;
			END_IF
			IF (intCmd = cFILE_HDL_CMD_NEW_FILE) OR (intCmd = cFILE_HDL_CMD_WRITE)THEN
				uinStep := cStep_FileWrite; // refresh actual file list
			ELSE
				intCmd := cFILE_HDL_CMD_DONE;
				uinStep := cStep_Wait4Job;
			END_IF
		ELSIF (uinSubStep = cSubStep_Error) THEN
			intCmd := cFILE_HDL_CMD_DONE;
			uinStep := cStep_Error;
		END_IF	
	
	cStep_FileWrite:	
		Out_strInfo := 'Write file busy';
		// entry action
		IF (uinStep<>uinStep_old) THEN
			Out_bolBusy := TRUE;
			uinSubStep := cSubStep_Done;
			uinStep_old := uinStep;
		END_IF	
		
		THIS^.M_FileWrite();
		
		IF (uinSubStep = cSubStep_Finished) THEN
			intCmd := cFILE_HDL_CMD_DONE;
			uinStep := cStep_FileClose;
		ELSIF (uinSubStep = cSubStep_Error) THEN
			intCmd := cFILE_HDL_CMD_DONE;
			uinStep := cStep_Error;
		END_IF
		
	cStep_FileClose:
		Out_strInfo := 'Close file busy';
		// entry action
		IF (uinStep<>uinStep_old) THEN	
			Out_bolBusy := TRUE;
			uinSubStep := cSubStep_Done;
			uinStep_old := uinStep;
		END_IF	
		
		THIS^.M_FileClose();
		
		IF (uinSubStep = cSubStep_Finished) THEN
			IF (intCmd = cFILE_HDL_CMD_NEW_FILE) OR (intCmd = cFILE_HDL_CMD_WRITE) THEN
				uinStep := cStep_NewFile;
			ELSE
				uinStep := cStep_Wait4Job;
			END_IF
			
		ELSIF (uinSubStep = cSubStep_Error) THEN
			intCmd := cFILE_HDL_CMD_DONE;
			uinStep := cStep_Error;
		END_IF	
		
	cStep_FileArchive:	
		// entry action
		Out_strInfo := 'Archive file busy';
		IF (uinStep<>uinStep_old) THEN	
			Out_bolBusy := TRUE;
			uinSubStep := cSubStep_Done;
			uinStep_old := uinStep;
			strPathNameArchive :=  THIS^.M_GetPathName(In_bolSufixDateTime:=TRUE,In_strSufixBeforeDateTime:=strSufixArchive);
		END_IF	

		// copy takes a lot of time!!! THIS^.M_FileCopy(In_strPathNameSrc := strPathName, In_strPathNameDst :=strPathNameArchive);
		THIS^.M_FileRename(In_strNetId := strNetId,In_strPathNewName:=strPathNameArchive,In_strPathOldName:=strPathName);
		
		IF (uinSubStep = cSubStep_Finished) THEN
			uinStep :=  cStep_FileOpen; // open "new file"// after copy delete original file cStep_FileDelete;
		ELSIF (uinSubStep = cSubStep_Error) THEN
			intCmd := cFILE_HDL_CMD_DONE;
			uinStep := cStep_Error;
		END_IF	
	
	cStep_Error:	
		// entry action
		IF (uinStep<>uinStep_old) THEN
			Out_strInfo := CONCAT(STR1:='Error - ',STR2:= Out_strInfo);
			Out_bolBusy := FALSE;
			uinStep_old := uinStep;
		END_IF
		
		
		IF (intCmd<>cFILE_HDL_CMD_DONE) THEN
			Out_udiErrId := 0;
			uinSubStep := cSubStep_Done;
			IF ( uin_FileHandle <> 0 ) THEN
				uinStep := cStep_FileClose; (* Close the source file *)
			ELSE
				uinStep := cStep_Wait4Job;
			END_IF
		END_IF	
				
END_CASE

PROPERTY PUBLIC ActFileSize : UDINT
GET
ActFileSize := LREAL_TO_UDINT(lreCurFileSize);
END_GET
END_PROPERTY

METHOD PUBLIC M_Cmd_FileDelete : BOOL
VAR_INPUT

END_VAR
intCmd := cFILE_HDL_CMD_FILE_DELETE;
END_METHOD

METHOD PUBLIC M_Cmd_NewFile : BOOL
VAR_INPUT

END_VAR
pWriteBuff := 0;
udiWriteLen := 0;
intCmd := cFILE_HDL_CMD_NEW_FILE;
END_METHOD

METHOD PUBLIC M_Cmd_WriteBuffer : BOOL
VAR_INPUT
	In_p_bytWriteBuff: POINTER TO BYTE;
	In_udiWriteLen : UDINT;
END_VAR
pWriteBuff := In_p_bytWriteBuff;
udiWriteLen := In_udiWriteLen;
intCmd := cFILE_HDL_CMD_WRITE;
END_METHOD

METHOD PROTECTED M_FileClose : BOOL
VAR_INPUT
	 
END_VAR
VAR
	strMyName : STRING := 'M_FileClose: ';
END_VAR
CASE uinSubStep OF
	cSubStep_Done:	
		Out_strInfo :=  CONCAT(CONCAT(Out_strInfo, strMyName) , 'start');
		
		fbFileClose_1.sNetId := fbFileOpen_1.sNetId;
		fbFileClose_1.hFile := uin_FileHandle;
		fbFileClose_1.tTimeout := T#3S;
		fbFileClose_1(bExecute:= FALSE);
		fbFileClose_1(bExecute:= TRUE);
		
		uinSubStep := 1;
		
	1: 
		Out_strInfo :=  CONCAT(CONCAT(Out_strInfo, strMyName) , 'busy');	

		(* wait until function block not busy *)
		fbFileClose_1( bExecute := FALSE );
		IF NOT fbFileClose_1.bBusy THEN
			uin_FileHandle := 0;
			IF NOT fbFileClose_1.bError THEN
				uinSubStep := cSubStep_Finished;
			ELSE 
				Out_udiErrId := fbFileClose_1.nErrID; // 0x703 	Invalid or unknown file handle., 0x70E 	File was opened with wrong method ( e.g. with 'obsolete' FILEOPEN function block ). 
				uinSubStep := cSubStep_Error;
			END_IF
		END_IF
		
	cSubStep_Finished: 
		// succesfully finished
		
	cSubStep_Error:
		Out_strInfo :=  CONCAT(CONCAT(Out_strInfo, strMyName) , CONCAT('error active - number:' , DWORD_TO_HEXSTR( fbFileClose_1.nErrID, 0, FALSE )));
		Out_udiErrId := fbFileClose_1.nErrID;
END_CASE
END_METHOD

METHOD PROTECTED M_FileCopy : BOOL
VAR_INPUT
	 In_strNetIdSrc : STRING(23);
	 In_strPathNameSrc : T_MaxString;
	 In_strNetIdDst : STRING(23);
	 In_strPathNameDst : T_MaxString;
END_VAR
VAR
	strMyName : STRING := 'M_FileCopy: ';
END_VAR
CASE uinSubStep OF
	cSubStep_Done:	
		Out_strInfo :=  CONCAT(CONCAT(Out_strInfo, strMyName) , 'start');
		
		fbFileCopy_1.srcNetId := In_strNetIdSrc; // only local access
		fbFileCopy_1.destNetId := In_strNetIdDst; // only local access
		fbFileCopy_1.srcFileName := In_strPathNameSrc;
		fbFileCopy_1.destFileName := In_strPathNameDst;
		fbFileCopy_1.tAdsTimeOut := T#3S;
		fbFileCopy_1(bExecute:= FALSE);
		fbFileCopy_1(bExecute:= TRUE);
		
		uinSubStep := 1;
		
	1: 
		Out_strInfo :=  CONCAT(CONCAT(Out_strInfo, strMyName) , 'busy');	

		(* wait until function block not busy *)
		fbFileCopy_1( bExecute := FALSE );
		IF NOT fbFileCopy_1.bBusy THEN
			uin_FileHandle := 0;
			IF NOT fbFileCopy_1.bError THEN
				uinSubStep := cSubStep_Finished;
			ELSE 
				Out_udiErrId := fbFileCopy_1.nErrID; 
				uinSubStep := cSubStep_Error;
			END_IF
		END_IF
		
	cSubStep_Finished: 
		// succesfully finished
		
	cSubStep_Error:
		Out_strInfo :=  CONCAT(CONCAT(Out_strInfo, strMyName) , CONCAT('error active - number:' , DWORD_TO_HEXSTR( fbFileCopy_1.nErrID, 0, FALSE )));
		Out_udiErrId := fbFileCopy_1.nErrID;
END_CASE
END_METHOD

METHOD PROTECTED M_FileDelete : BOOL
VAR_INPUT
	In_strNetId : STRING(23);
	In_strPathName : T_MaxString;  
END_VAR
VAR
	strMyName : STRING := 'M_FileDelete: ';
END_VAR

CASE uinSubStep OF
	cSubStep_Done:	
		Out_strInfo :=  CONCAT(CONCAT(Out_strInfo, strMyName) , 'start');
		
		fbFileDelete_1.sNetId :=In_strNetId;
		fbFileDelete_1.sPathName := In_strPathName;
		fbFileDelete_1.ePath := PATH_GENERIC;
		fbFileDelete_1.tTimeout := T#3S;
		fbFileDelete_1(bExecute:= FALSE);
		fbFileDelete_1(bExecute:= TRUE);
		
		uinSubStep := 1;
		
	1: 
		Out_strInfo :=  CONCAT(CONCAT(Out_strInfo, strMyName) , 'busy');	

		(* wait until function block not busy *)
		fbFileDelete_1( bExecute := FALSE );
		IF NOT fbFileDelete_1.bBusy THEN
			IF NOT fbFileDelete_1.bError THEN
				uinSubStep := cSubStep_Finished;
			ELSE 
				Out_udiErrId := fbFileDelete_1.nErrID;
				uinSubStep := cSubStep_Error;
			END_IF
		END_IF
		
	cSubStep_Finished: 
		// succesfully finished
		
	cSubStep_Error:
		Out_strInfo :=  CONCAT(CONCAT(Out_strInfo, strMyName) , CONCAT('error active - number:' , DWORD_TO_HEXSTR( fbFileDelete_1.nErrID, 0, FALSE )));
		Out_udiErrId := fbFileDelete_1.nErrID;
END_CASE
END_METHOD

METHOD PROTECTED M_FileOpen : BOOL
VAR_INPUT
	In_strNetId : STRING(23);
	In_strPathName : T_MaxString;  
END_VAR
VAR
	strMyName : STRING := 'M_FileOpen: ';
END_VAR
CASE uinSubStep OF
	cSubStep_Done:	
		Out_strInfo :=  CONCAT(CONCAT(Out_strInfo, strMyName) , 'start');
		
		fbFileOpen_1.sNetId := In_strNetId;
		fbFileOpen_1.sPathName := In_strPathName;
		fbFileOpen_1.nMode := FOPEN_MODEAPPEND OR FOPEN_MODEPLUS OR FOPEN_MODEBINARY;      // "a+": Opens for reading and appending; the appending operation includes the removal of the EOF marker before new data is written to the file and the EOF marker is restored after writing is complete; creates the file first if it doesn’t exist.
																					// When a file is opened with the "a" or "a+" access type, all write operations occur at the end of the file. The file pointer can be repositioned using FB_FileSeek, but is always moved back to the end of the file before any write operation is carried out. Thus, existing data cannot be overwritten.                       

		fbFileOpen_1.ePath := PATH_GENERIC;
		fbFileOpen_1.tTimeout := T#3S;
		fbFileOpen_1(bExecute:= FALSE);
		fbFileOpen_1(bExecute:= TRUE);
		
		uinSubStep := 1;
		
	1: 
		Out_strInfo :=  CONCAT(CONCAT(Out_strInfo, strMyName) , 'busy');	

		(* wait until function block not busy *)
		fbFileOpen_1( bExecute := FALSE );
		IF NOT fbFileOpen_1.bBusy THEN
			uin_FileHandle := fbFileOpen_1.hFile;
			IF NOT fbFileOpen_1.bError THEN
				uinSubStep := cSubStep_Finished;
			ELSE 
				Out_udiErrId := fbFileOpen_1.nErrID;
				uinSubStep := cSubStep_Error;
			END_IF
		END_IF
		
	cSubStep_Finished: 
		// succesfully finished
		
	cSubStep_Error:
		Out_strInfo :=  CONCAT(CONCAT(Out_strInfo, strMyName) , CONCAT('error active - number:' , DWORD_TO_HEXSTR( fbFileOpen_1.nErrID, 0, FALSE )));
		Out_udiErrId := fbFileOpen_1.nErrID;
END_CASE
END_METHOD

METHOD PROTECTED M_FileRename : BOOL
VAR_INPUT
	 In_strNetId : STRING(23);
	 In_strPathOldName : T_MaxString;
	 In_strPathNewName : T_MaxString;
END_VAR
VAR
	strMyName : STRING := 'M_FileRename: ';
END_VAR
CASE uinSubStep OF
	cSubStep_Done:	
		Out_strInfo :=  CONCAT(CONCAT(Out_strInfo, strMyName) , 'start');
		
		fbFileRename_1.sNetId := In_strNetId;
		fbFileRename_1.sOldName := In_strPathOldName;
		fbFileRename_1.sNewName := In_strPathNewName;
		fbFileRename_1.ePath := PATH_GENERIC;
		fbFileRename_1.tTimeout := T#3S;
		fbFileRename_1(bExecute:= FALSE);
		fbFileRename_1(bExecute:= TRUE);
		
		uinSubStep := 1;
		
	1: 
		Out_strInfo :=  CONCAT(CONCAT(Out_strInfo, strMyName) , 'busy');	

		(* wait until function block not busy *)
		fbFileRename_1( bExecute := FALSE );
		IF NOT fbFileRename_1.bBusy THEN
			IF NOT fbFileRename_1.bError THEN
				uinSubStep := cSubStep_Finished;
			ELSE 
				Out_udiErrId := fbFileRename_1.nErrID;
				uinSubStep := cSubStep_Error;
			END_IF
		END_IF
		
	cSubStep_Finished: 
		// succesfully finished
		
	cSubStep_Error:
		Out_strInfo :=  CONCAT(CONCAT(Out_strInfo, strMyName) , CONCAT('error active - number:' , DWORD_TO_HEXSTR( fbFileRename_1.nErrID, 0, FALSE )));
		Out_udiErrId := fbFileRename_1.nErrID;
END_CASE
END_METHOD

METHOD PROTECTED M_FileWrite : BOOL
VAR_INPUT
	 
END_VAR
VAR
	strMyName : STRING := 'M_FileClose: ';
END_VAR
CASE uinSubStep OF
	cSubStep_Done:	
		Out_strInfo :=  CONCAT(CONCAT(Out_strInfo, strMyName) , 'start');
		
		fbFileWrite_1.sNetId := fbFileOpen_1.sNetId;
		fbFileWrite_1.hFile := uin_FileHandle; // file handle from file open
		fbFileWrite_1.pWriteBuff := pWriteBuff; // Write buffer adress
		fbFileWrite_1.cbWriteLen := udiWriteLen; // Write buffer len
		fbFileWrite_1.tTimeout := T#3S;
		fbFileWrite_1(bExecute:= FALSE);
		fbFileWrite_1(bExecute:= TRUE);
		
		uinSubStep := 1;
		
	1: 
		Out_strInfo :=  CONCAT(CONCAT(Out_strInfo, strMyName) , 'busy');	

		(* wait until function block not busy *)
		fbFileWrite_1( bExecute := FALSE );
		IF NOT fbFileWrite_1.bBusy THEN
			lreCurFileSize := lreCurFileSize + fbFileWrite_1.cbWrite;
			IF NOT fbFileWrite_1.bError THEN
				uinSubStep := cSubStep_Finished;
			ELSE 
				Out_udiErrId := fbFileWrite_1.nErrID; // 0x703 	Invalid or unknown file handle., 0x70E 	File was opened with wrong method ( e.g. with 'obsolete' FILEOPEN function block ). 
				uinSubStep := cSubStep_Error;
			END_IF
		END_IF
		
	cSubStep_Finished: 
		// succesfully finished
		
	cSubStep_Error:
		Out_strInfo :=  CONCAT(CONCAT(Out_strInfo, strMyName) , CONCAT('error active - number:' , DWORD_TO_HEXSTR( fbFileWrite_1.nErrID, 0, FALSE )));
		Out_udiErrId := fbFileOpen_1.nErrID;
END_CASE
END_METHOD

METHOD PRIVATE M_GetPathName : T_MaxString
VAR_INPUT
	In_strSufixBeforeDateTime : T_MaxString;
	In_bolSufixDateTime : BOOL;
END_VAR
VAR
	strTemp: Tc2_System.T_MaxString;
	strTempDateTime: Tc2_System.T_MaxString;
END_VAR

//strPathName := CONCAT(CONCAT(CONCAT(CONCAT(strPath , '\') , strFileName ), '.' ), strFileExt);


strTemp := strPath; //CONCAT(strPath , '\');
strTemp := CONCAT(strTemp , strFileName);
strTemp := CONCAT(strTemp , In_strSufixBeforeDateTime);
IF (In_bolSufixDateTime = TRUE) THEN
	strTempDateTime := '';
	strTempDateTime := CONCAT(strTempDateTime , WORD_TO_STRING(fbNT_GetTime.TIMESTR.wYear));
	IF (fbNT_GetTime.TIMESTR.wMonth<10) THEN
		strTempDateTime := CONCAT(strTempDateTime , '0');
	END_IF
	strTempDateTime := CONCAT(strTempDateTime , WORD_TO_STRING(fbNT_GetTime.TIMESTR.wMonth));
	IF (fbNT_GetTime.TIMESTR.wDay<10) THEN
		strTempDateTime := CONCAT(strTempDateTime , '0');
	END_IF
	strTempDateTime := CONCAT(strTempDateTime , WORD_TO_STRING(fbNT_GetTime.TIMESTR.wDay));
	strTempDateTime := CONCAT(strTempDateTime , '_');
	IF (fbNT_GetTime.TIMESTR.wHour<10) THEN
		strTempDateTime := CONCAT(strTempDateTime , '0');
	END_IF
	strTempDateTime := CONCAT(strTempDateTime , WORD_TO_STRING(fbNT_GetTime.TIMESTR.wHour));
	IF (fbNT_GetTime.TIMESTR.wMinute<10) THEN
		strTempDateTime := CONCAT(strTempDateTime , '0');
	END_IF
	strTempDateTime := CONCAT(strTempDateTime , WORD_TO_STRING(fbNT_GetTime.TIMESTR.wMinute));
	IF (fbNT_GetTime.TIMESTR.wSecond<10) THEN
		strTempDateTime := CONCAT(strTempDateTime , '0');
	END_IF
	strTempDateTime := CONCAT(strTempDateTime , WORD_TO_STRING(fbNT_GetTime.TIMESTR.wSecond));
	strTemp := CONCAT(strTemp , strTempDateTime);
END_IF
strTemp := CONCAT(strTemp , '.');
M_GetPathName := CONCAT(strTemp , strFileExt);
END_METHOD

METHOD PUBLIC M_Init : BOOL
VAR_INPUT
	In_strNetId: STRING(23); // NetId to write to foreign system drives
	IN_strPath : Tc2_System.T_MaxString; 	// Contains only the path 
	IN_strFileName : Tc2_System.T_MaxString;// Contains only the filename
	IN_strFileExt : Tc2_System.T_MaxString;	// Contains only the ext
	IN_uinMaxNrOfFilesInFolder:UINT; // max number of files in folder
	IN_timFileSupervisionPeriod : TIME;// time periode for checking max file nuimber in folder
	IN_lreMaxFileSize : LREAL;// maximal allowed filesize for file -> archivate and deleter or create new
	
END_VAR
strNetId := In_strNetId;
strPath := IN_strPath;
strFileName := IN_strFileName;
strFileExt := IN_strFileExt;
lreMaxFileSize := IN_lreMaxFileSize; // maximal allowed filesize for file -> archivate and deleter or create new

fbFolderHdl_1.M_INIT(IN_strPath := strPath,IN_strPrefixFileName:=strFileName,IN_strFileExt:=strFileExt,In_strNetId:=strNetId);
fbFolderHdl_1.MaxNrOfFilesInFolder := IN_uinMaxNrOfFilesInFolder;
fbFolderHdl_1.FileSupervisionPeriod := IN_timFileSupervisionPeriod;
bolInitDone := TRUE;
END_METHOD

END_FUNCTION_BLOCK

// POUs/Utility/FileFolder/FB_FolderHdl
FUNCTION_BLOCK FB_FolderHdl

VAR_OUTPUT
	Out_bolBusy : BOOL; // busy
	Out_udiErrId : UDINT; // error id
	Out_strInfo : STRING; //
	Out_bolInitDone: BOOL;
END_VAR
VAR
	uinStep: UINT;
	uinStep_old : UINT;
	uinSubStep : UINT;
	intCmd : INT;
	bolInitDone : BOOL;
	bolFileNrExceedArraySize : BOOL; // more than max possibel managed files found -> delete in cyclic
	// configurations/parameters
	strNetId : STRING(23);
	strPath : T_MaxString; 	// Contains only the path 
	strPathName : T_MaxString; 	// Contains the whole search expresion
	strFilePrefix : T_MaxString;	// Contains only the filename
	strFileExt : T_MaxString;	// Contains only the ext
	strTemp : T_MaxString;
	timFileSupervisionPeriod : TIME;
	uinMaxNrOfFilesInFolder : UINT; // max number of files in folder defined
	
	lreTotalFileSize : LREAL;
	aFileList : ARRAY[1..cFILE_HDL_MAX_NR_OF_FILE_TO_MANAGE]  OF ST_FindFileEntry;
	bolAbort : BOOL;
	intOldestFile : INT := 1; // sort list oldest =1
	udiNrOfFilesInFolder : UDINT;

	fbEnumFindFileList_1 : FB_EnumFindFileList;
	fbFileDelete_1 : FB_FileDelete;
	fTON_1 : TON;
	
END_VAR
VAR CONSTANT
	// specific steps definitions
	cStep_Start: UINT := 501;
	cStep_FileDelete: UINT := 100;
	cStep_Refresh: UINT := 101;
	cStep_Wait4Job: UINT := 500;
	cStep_Error: UINT := 256;
	
	cSubStep_Done: UINT := 0;
	cSubStep_Finished: UINT := 100;
	cSubStep_Error: UINT := 256;
	
	
	// commandes constants
	cFOLDER_HDL_CMD_DONE : INT := -1;
	cFOLDER_HDL_CMD_REFRESH_FILE_LIST : INT := 1;
END_VAR

(*__________________________________________________________________________________________________
¦	
¦	Vistaprint Schweiz GmbH
¦	CH - 8401 Winterthur
¦
¦	www.vistaprint.ch - info@vistaprint.ch
¦___________________________________________________________________________________________________

Function desription:
	Manage folder: 
	- Refresh list of files in specific folder
	- sort list form oldest to newest file
	- cyclic supervision of max number of files in folder
	- triggered supervision of max number of files in folder 
		
History:
Version		Date			Author		Comment
---------------------------------------------------------------------------------------------------
0.00.1		14.05.2014		AVME/KVO	Start history
___________________________________________________________________________________________________*)



CASE uinStep OF
	0:	
		// entry action
		IF (uinStep<>uinStep_old) THEN
			Out_strInfo := 'Wait for init ok -> call methode M_INIT()';
			uinSubStep := cSubStep_Done;
			uinStep_old := uinStep;
		END_IF
		
		IF bolInitDone THEN
			uinStep := cStep_Start;
		END_IF
		
	cStep_Start: 
		// entry action
		IF (uinStep<>uinStep_old) THEN
			Out_strInfo := 'Start';	
			Out_bolBusy := 0;
			Out_udiErrId := 0;
			uinSubStep := cSubStep_Done;
			fTON_1.IN := FALSE;
			fTON_1();
			uinStep_old := uinStep;
		END_IF
		
		intCmd := cFOLDER_HDL_CMD_REFRESH_FILE_LIST;// refresh actual file list first

		uinStep := cStep_Wait4Job;
		
	cStep_Wait4Job:	
		// entry action
		IF (uinStep<>uinStep_old) THEN
			Out_strInfo := 'Wait for job';
			Out_bolBusy := FALSE;
			uinSubStep := cSubStep_Done;
			uinStep_old := uinStep;
		END_IF

		IF (timFileSupervisionPeriod>T#0MS) THEN
			fTON_1.PT := timFileSupervisionPeriod;
			fTON_1.IN := TRUE;
			fTON_1();
		END_IF
		
		IF (intCmd = cFOLDER_HDL_CMD_REFRESH_FILE_LIST) OR (fTON_1.Q=TRUE) THEN
			uinStep := cStep_Refresh; // refresh actual file list
		ELSE
			IF (udiNrOfFilesInFolder>uinMaxNrOfFilesInFolder) AND (uinMaxNrOfFilesInFolder<>0) THEN
				intOldestFile := 1; // first entry
				uinStep := cStep_FileDelete;
			END_IF
		END_IF
		
		

	cStep_Refresh:	
		// entry action
		IF (uinStep<>uinStep_old) THEN
			Out_strInfo := 'Refresh file list busy';
			Out_bolBusy := TRUE;
			fTON_1.IN := FALSE;
			fTON_1();
			uinSubStep := cSubStep_Done;
			uinStep_old := uinStep;
		END_IF

		THIS^.M_RefreshFileList();
		
		IF (uinSubStep = cSubStep_Finished) THEN
			THIS^.M_SortFileList();
			intCmd := cFOLDER_HDL_CMD_DONE;
			Out_bolInitDone := TRUE; // valid file list
			uinStep := cStep_Wait4Job;
		ELSIF (uinSubStep = cSubStep_Error) THEN
			intCmd := cFOLDER_HDL_CMD_DONE;
			uinStep := cStep_Error;
		END_IF	

	cStep_FileDelete:
	// entry action
		IF (uinStep<>uinStep_old) THEN
			Out_strInfo := 'Delete file busy';
			Out_bolBusy := TRUE;
			uinSubStep := cSubStep_Done;
			uinStep_old := uinStep;
		END_IF	
		
		strTemp := strPath;
		strTemp := CONCAT(strTemp , aFileList[intOldestFile].sFileName);
		THIS^.M_FileDelete(strTemp);
		
		IF (uinSubStep = cSubStep_Finished) THEN
			intCmd := cFOLDER_HDL_CMD_DONE;
			uinStep := cStep_Refresh; 
		ELSIF (uinSubStep = cSubStep_Error) THEN
			intCmd := cFOLDER_HDL_CMD_DONE;
			uinStep := cStep_Error;
		END_IF
		
	cStep_Error:	
		// entry action
		IF (uinStep<>uinStep_old) THEN
			// written in sub Out_strInfo := 'Error';
			Out_bolBusy := FALSE;
			uinStep_old := uinStep;
		END_IF
		
		IF (intCmd<>cFOLDER_HDL_CMD_DONE) THEN
			Out_udiErrId := 0;
			uinSubStep := cSubStep_Done;
			uinStep := cStep_Wait4Job;
		END_IF
END_CASE

PROPERTY PUBLIC FileSupervisionPeriod : TIME
GET
FileSupervisionPeriod := timFileSupervisionPeriod;
END_GET
SET
timFileSupervisionPeriod := FileSupervisionPeriod;
END_SET
END_PROPERTY

PROPERTY PUBLIC get_FileList : ARRAY[1..cFILE_HDL_MAX_NR_OF_FILE_TO_MANAGE]  OF ST_FindFileEntry;
GET
uinSubStep := 0;

WHILE (THIS^.M_RefreshFileList()=FALSE) DO
	//wait until read all files in folder
END_WHILE

THIS^.M_SortFileList(); // sort last write date -> oldest at position 1!
END_GET
END_PROPERTY

PROPERTY get_NewestFileEntry : ST_FindFileEntry
GET
uinSubStep := 0;
(* läuft nicvht???
WHILE (THIS^.M_RefrehFileList()=FALSE) DO
	//wait until read all files in folder
END_WHILE

THIS^.M_SortFileList(); // sort last write date -> oldest at position 1!
*)
get_NewestFileEntry := aFileList[udiNrOfFilesInFolder];
END_GET
END_PROPERTY

METHOD PUBLIC M_Cmd_RefreshFileList : BOOL
intCmd := cFOLDER_HDL_CMD_REFRESH_FILE_LIST;
END_METHOD

METHOD PROTECTED M_FileDelete : BOOL
VAR_INPUT
	strPathName : T_MaxString;  
END_VAR
VAR
	strMyName : STRING := 'M_FileDelete: ';
END_VAR

CASE uinSubStep OF
	cSubStep_Done:	
		Out_strInfo :=  CONCAT(CONCAT(Out_strInfo, strMyName) , 'start');
		
		fbFileDelete_1.sNetId := strNetId;
		fbFileDelete_1.sPathName := strPathName;
		fbFileDelete_1.ePath := PATH_GENERIC;
		fbFileDelete_1.tTimeout := T#3S;
		fbFileDelete_1(bExecute:= FALSE);
		fbFileDelete_1(bExecute:= TRUE);
		
		uinSubStep := 1;
		
	1: 
		Out_strInfo :=  CONCAT(CONCAT(Out_strInfo, strMyName) , 'busy');	

		(* wait until function block not busy *)
		fbFileDelete_1( bExecute := FALSE );
		IF NOT fbFileDelete_1.bBusy THEN
			IF NOT fbFileDelete_1.bError THEN
				uinSubStep := cSubStep_Finished;
			ELSE 
				Out_udiErrId := fbFileDelete_1.nErrID;
				uinSubStep := cSubStep_Error;
			END_IF
		END_IF
		
	cSubStep_Finished: 
		// succesfully finished
		
	cSubStep_Error:
		Out_strInfo :=  CONCAT(CONCAT(Out_strInfo, strMyName) , CONCAT('error active - number:' , DWORD_TO_HEXSTR( fbFileDelete_1.nErrID, 0, FALSE )));
		Out_udiErrId := fbFileDelete_1.nErrID;
END_CASE
END_METHOD

METHOD PUBLIC M_FileExist : BOOL
VAR_INPUT
	strPathName : Tc2_System.T_MaxString;
END_VAR
VAR
	fbEnum : FB_EnumFindFileEntry := ( sNetID := '', tTimeout := T#5S, sPathName := strPathName );
	uinState : UINT:=0;
END_VAR
WHILE (uinState<>10) DO
	CASE uinState OF
	0:
		fbEnum.sNetId := strNetId;
		fbEnum.eCmd := eEnumCmd_First; (* enum first entry *)
		uinState := 1;
	
	1: (* enum one entry *)
		fbEnum( bExecute := FALSE );
		fbEnum( bExecute := TRUE );
		uinState := 2;
	
	2: (* wait until function block not busy *)
		fbEnum( bExecute := FALSE );
		IF NOT fbEnum.bBusy THEN
			IF NOT fbEnum.bError THEN
				IF NOT fbEnum.bEOE THEN
					M_FileExist := TRUE;
					EXIT;
				ELSE (* no more entries *)
					M_FileExist := FALSE;
					EXIT;
				END_IF
			ELSE (* log error *)
				M_FileExist := FALSE;
				EXIT;
			END_IF
		END_IF
	END_CASE
END_WHILE
END_METHOD

METHOD M_getFileInfo : ST_FindFileEntry
VAR_INPUT
	IN_strFileNameWithExt : Tc2_System.T_MaxString;// Contains the filename with extension
END_VAR
VAR
	ii : UDINT;
	udiUpperLimit : UDINT;
END_VAR
IF (udiNrOfFilesInFolder<cFILE_HDL_MAX_NR_OF_FILE_TO_MANAGE) THEN
	udiUpperLimit := udiNrOfFilesInFolder;
ELSE
	udiUpperLimit := cFILE_HDL_MAX_NR_OF_FILE_TO_MANAGE;	
END_IF

FOR ii:= 0 TO udiUpperLimit DO
	IF (FIND(aFileList[ii].sFileName,IN_strFileNameWithExt)<>0) THEN
		M_getFileInfo := aFileList[ii];
		EXIT;
	END_IF
END_FOR
END_METHOD

METHOD PUBLIC M_GetFileSize : LREAL
VAR_INPUT
	In_strFileName: T_MaxString;
END_VAR
VAR
	i:UDINT;
END_VAR
IF (udiNrOfFilesInFolder=0) THEN
	WHILE (THIS^.M_RefreshFileList()=FALSE) DO
		//wait until read all files in folder
	END_WHILE
END_IF

M_GetFileSize := 0.0;

FOR i := 1 TO udiNrOfFilesInFolder BY 1 DO
	IF (In_strFileName = aFileList[i].sFileName) THEN
		M_GetFileSize := Tc2_Utilities.UINT64_TO_LREAL(aFileList[i].fileSize);
		EXIT;
	END_IF
END_FOR;
END_METHOD

METHOD PUBLIC M_Init : BOOL
VAR_INPUT
	IN_strPath : Tc2_System.T_MaxString; 	// Contains only the path 
	IN_strPrefixFileName : Tc2_System.T_MaxString;// Contains only the filename
	IN_strFileExt : Tc2_System.T_MaxString;	// Contains only the ext
	In_strNetId: STRING(23); // NetId to write to foreign system drives
END_VAR
VAR
	strTemp: Tc2_System.T_MaxString;
END_VAR
strNetId := In_strNetId;
strPath := IN_strPath;
strFilePrefix := IN_strPrefixFileName;
strFileExt := IN_strFileExt;
strTemp := strPath;//todo check path allready added / CONCAT(strPath , '\');
strTemp := CONCAT(strTemp , strFilePrefix);
IF (strFileExt='') THEN
	strPathName := strTemp;
ELSE
	strTemp := CONCAT(strTemp , '.');
	strPathName := CONCAT(strTemp , strFileExt);
END_IF
uinStep := 0;
bolInitDone := TRUE;
END_METHOD

METHOD PUBLIC M_RefreshFileList : BOOL
VAR
	strMyName : STRING := 'M_RefrehFileList: ';
	strTemp : STRING;
END_VAR
CASE uinSubStep OF
	cSubStep_Done:	
		Out_strInfo :=  CONCAT(CONCAT(Out_strInfo, strMyName) , 'start');
		
		M_RefreshFileList := FALSE;
		udiNrOfFilesInFolder := 0;
		
		// define proberties for searching files in folder
		fbEnumFindFileList_1.sNetId := strNetId;

		strTemp := strPath;//todo check path allready added / CONCAT(strPath , '\');
		strTemp := CONCAT(strTemp , strFilePrefix);
		IF (strFileExt='') THEN
			strTemp := CONCAT(strTemp , '*'); // all data types
		ELSE
			strTemp := CONCAT(strTemp , '*.');
			strTemp := CONCAT(strTemp , strFileExt);
		END_IF

		fbEnumFindFileList_1.sPathName := strTemp; // read all files in the defined folder with the defined extension
        fbEnumFindFileList_1.pFindList := ADR(aFileList);
        fbEnumFindFileList_1.cbFindList := SIZEOF(aFileList);
        fbEnumFindFileList_1.tTimeout := DEFAULT_ADS_TIMEOUT;
		fbEnumFindFileList_1.eCmd := E_EnumCmdType.eEnumCmd_First;	(* enum first entry *)
		uinSubStep := 1;
		
	1: 
		Out_strInfo :=  CONCAT(CONCAT(Out_strInfo, strMyName) , 'Reading files in folder busy');	
		
		(* enum one entry *)
		IF bolAbort THEN
			bolAbort := FALSE;
			fbEnumFindFileList_1.eCmd := E_EnumCmdType.eEnumCmd_Abort;
		END_IF
		
		fbEnumFindFileList_1( bExecute := FALSE );
		fbEnumFindFileList_1( bExecute := TRUE );
		uinSubStep := 2;
		
	2:	
		Out_strInfo := CONCAT(CONCAT(Out_strInfo, strMyName) , 'Reading files in folder busy');	
		
		(* wait until function block not busy *)
		fbEnumFindFileList_1( bExecute := FALSE );
		IF NOT fbEnumFindFileList_1.bBusy THEN
			udiNrOfFilesInFolder := fbEnumFindFileList_1.nFindFiles;
			IF NOT fbEnumFindFileList_1.bError THEN
				IF NOT fbEnumFindFileList_1.bEOE THEN
					bolFileNrExceedArraySize := TRUE;
					(* read more informations -> not meaningful 
					fbEnumFindFileList_1.eCmd := E_EnumCmdType.eEnumCmd_Next; (* enum next entry *)
					uinSubStep := 1;*)
					uinSubStep := cSubStep_Finished; // reduce maximum in cyclic actions...-> delete if > max 
				ELSE (* no more entries *)
					uinSubStep := cSubStep_Finished;
				END_IF
			ELSE (* log error *)
				Out_udiErrId := fbEnumFindFileList_1.nErrID;
				uinSubStep := cSubStep_Error;
			END_IF
		END_IF

	cSubStep_Finished: 
		// succesfully finished
		M_RefreshFileList := TRUE;
	cSubStep_Error:
		Out_strInfo :=  CONCAT(CONCAT(Out_strInfo, strMyName) , CONCAT('error active - number:' , DWORD_TO_HEXSTR( fbEnumFindFileList_1.nErrID, 0, FALSE )));
		Out_udiErrId := fbEnumFindFileList_1.nErrID;
		M_RefreshFileList := TRUE;
END_CASE
END_METHOD

METHOD PUBLIC M_SortFileList : BOOL
VAR_INPUT

END_VAR
VAR
	stTempFile 	: ST_FindFileEntry;
	bolNoChangeDone: BOOL;
	i,j :UDINT;
END_VAR
// BubbleSort
M_SortFileList := FALSE;

IF (udiNrOfFilesInFolder>1) THEN
	lreTotalFileSize := UINT64_TO_LREAL(aFileList[1].fileSize);
	FOR i := 1 TO udiNrOfFilesInFolder BY 1 DO
		bolNoChangeDone := TRUE;
		FOR j := 1 TO (udiNrOfFilesInFolder-i) BY 1 DO
			IF (i=1) THEN// count total filesize
				lreTotalFileSize := lreTotalFileSize + Tc2_Utilities.UINT64_TO_LREAL(aFileList[j+1].fileSize);
			END_IF
			
			IF (FILETIME_TO_DT(aFileList[j].lastWriteTime) > FILETIME_TO_DT(aFileList[j + 1].lastWriteTime)) THEN
				// swap files
				memcpy(ADR(stTempFile), ADR(aFileList[j]),SIZEOF(stTempFile));
				memcpy(ADR(aFileList[j]), ADR(aFileList[j + 1]),SIZEOF(stTempFile));
				memcpy(ADR(aFileList[j + 1]), ADR(stTempFile),SIZEOF(stTempFile));
				bolNoChangeDone := FALSE; // at least one change done
			END_IF
			
		END_FOR; 
		IF (bolNoChangeDone) THEN
			EXIT;
		END_IF
	END_FOR;
END_IF;
M_SortFileList := TRUE;
END_METHOD

PROPERTY MaxNrOfFilesInFolder : UINT
GET
MaxNrOfFilesInFolder := uinMaxNrOfFilesInFolder;
END_GET
SET
// not more files allowed as defined in struct....Sort problem
IF (MaxNrOfFilesInFolder<cFILE_HDL_MAX_NR_OF_FILE_TO_MANAGE) THEN
	uinMaxNrOfFilesInFolder := MaxNrOfFilesInFolder;
ELSE
	uinMaxNrOfFilesInFolder := UDINT_TO_UINT(cFILE_HDL_MAX_NR_OF_FILE_TO_MANAGE-1);	
END_IF
END_SET
END_PROPERTY

END_FUNCTION_BLOCK

// POUs/Utility/Logger/BasLog/FB_BasLogTest_Client
FUNCTION_BLOCK FB_BasLogTest_Client
VAR_INPUT
	In_p_fbBasLog: POINTER TO FB_BasLog; // only one central FB_BasLog instance allowed per PLC!!!
END_VAR
VAR_OUTPUT
END_VAR
VAR
	stData : T_Bl_BaseStruc;
	bolInit : BOOL := FALSE;
	pReadHandle : POINTER TO POINTER TO T_Queue_Info;
	uinInitStatus : UINT;
	uinChangeMaskStatus :UINT;
	uinReadStatus : UINT;
	bolChangeMask : BOOL;
	bolRead : BOOL;
	fbTimeStamp: FB_TimeStamp;
END_VAR

(*__________________________________________________________________________________________________
¦	
¦	Vistaprint Schweiz GmbH
¦	CH - 8401 Winterthur
¦
¦	www.vistaprint.ch - info@vistaprint.ch
¦___________________________________________________________________________________________________

Function desription:
Example and test programm for testing the base log system - read data from base log

History:
Version		Date			Author		Comment
---------------------------------------------------------------------------------------------------
0.00.1		14.07.2014		AVME/KVO	Start history
___________________________________________________________________________________________________*)

// system init onetime after start up
IF (bolInit=FALSE) THEN
	// init timer system
	fbTimeStamp.In_strNetId := ''; // use local system time
	fbTimeStamp.In_t_CycleTimeRefreshTimeZone := T#15M; // cyclic check time zone settings
	//init baselog system, one time should be called per baslog system
	In_p_fbBasLog^.M_ClientInit(In_strClientName:='BaseLog',In_udiMask := 16#FFFFFFFF, In_uinNrOfElement:= 128,In_p_fbTimeStamp:=ADR(fbTimeStamp),In_bolUseLocalTimeStamp:=TRUE,Out_pHandle=>pReadHandle,Out_uinStatus=>uinInitStatus);
	
	bolInit := TRUE;
END_IF

fbTimeStamp(); // cyclic call needed for valid time stamp / synchronisation
	
(* change mak on runtime *)
IF (bolRead = TRUE) THEN
	(* cyclically read out of data*)
	uinReadStatus:= In_p_fbBasLog^.M_Read(In_pHandle:=pReadHandle,In_pData:=ADR(stData)); 
END_IF

(* change mak on runtime *)
IF (bolChangeMask = TRUE) THEN
	uinChangeMaskStatus := In_p_fbBasLog^.M_ChangeMask(In_strClientName:='BaseLog',In_udiNewMask:= 16#0F0F0F0F);
	bolChangeMask := FALSE;
END_IF

END_FUNCTION_BLOCK

// POUs/Utility/Logger/BasLog/FB_BasLogTest_Sender
FUNCTION_BLOCK FB_BasLogTest_Sender
VAR_INPUT
	In_p_fbBasLog: POINTER TO FB_BasLog; // only one central FB_BasLog instance allowed per PLC!!!
END_VAR
VAR_OUTPUT
END_VAR
VAR
	bolInit : BOOL := FALSE;
	pHandle : POINTER TO T_Bl_LibHandleRow;
	uinGetHandleStatus : UINT;
	uinWriteStatus :UINT;
	uinDoWrite : UINT;
	dinPar1 : DINT;
	strText1 : STRING(30):='Controller 1';
	strText2 : STRING(30):='Alarm sub info';
END_VAR

(*__________________________________________________________________________________________________
¦	
¦	Vistaprint Schweiz GmbH
¦	CH - 8401 Winterthur
¦
¦	www.vistaprint.ch - info@vistaprint.ch
¦___________________________________________________________________________________________________

Function desription:
Example and test programm for testing the queue system - write data to base log

History:
Version		Date			Author		Comment
---------------------------------------------------------------------------------------------------
0.00.1		14.07.2014		AVME/KVO	Start history
___________________________________________________________________________________________________*)

// system init onetime after start up
IF (bolInit=FALSE) THEN
	uinGetHandleStatus := In_p_fbBasLog^.M_GetHandle(Out_pHandle=>pHandle);
	
	bolInit := TRUE;
END_IF

// write base log entries
IF (uinDoWrite>0) THEN
	uinDoWrite := uinDoWrite - 1;
	dinPar1 := dinPar1 + 1;
	uinWriteStatus := In_p_fbBasLog^.M_Log(In_pHandle:=pHandle,In_udiLogType:=BasLog.cLOGTYPE_ALARM,In_intCtrlID:=11,In_strText1:=strText1,In_strText2:=strText2,In_dinPar1:=dinPar1,In_dinPar2:=0,In_dinPar3:=0,In_dinPar4:=0) ;
END_IF

END_FUNCTION_BLOCK

// POUs/Utility/Logger/DatLog/FB_DatLog
FUNCTION_BLOCK FB_DatLog
VAR_INPUT
END_VAR
VAR_OUTPUT
END_VAR
VAR
	stDatLogLibInfo : T_DL_LibInfo;
	fbPLC_ReadSymInfo: PLC_ReadSymInfoByNameEx; // only one init allowed on the same time....
END_VAR

(*__________________________________________________________________________________________________
¦	
¦	Vistaprint Schweiz GmbH
¦	CH - 8401 Winterthur
¦
¦	www.vistaprint.ch - info@vistaprint.ch
¦___________________________________________________________________________________________________

Function desription:
Base logger system. The FUB must be called defined globally one time in PLC-program. After that the implemented 
sender and receiver must interact over the public methodes of the FB_BasLog.

History:
Version		Date			Author		Comment
---------------------------------------------------------------------------------------------------
0.00.1		14.07.2014		AVME/KVO	Start history
___________________________________________________________________________________________________*)

METHOD PROTECTED M_AllocMEM : POINTER TO BYTE

VAR_INPUT
	In_SizeOfBuffer : UINT; // Byte size of quee to allocate
END_VAR
// Debug counter
M_AllocMEM := __NEW(BYTE,In_SizeOfBuffer);

// check if allocate memory is ok
IF (M_AllocMEM=TC3_MEMMAN.NULL) THEN
	M_AllocMEM := TC3_MEMMAN.NULL;
ELSE
	Tc2_System.MEMSET(M_AllocMEM,0,In_SizeOfBuffer); // init with zero.
END_IF
END_METHOD

METHOD PRIVATE M_CheckAndAppendDatLogInfo : Pointer TO T_DL_SysInfo
VAR_INPUT
	In_strDatLogName: STRING(DatLog.cMAX_SYS_NAME_LENGTH); // name of the client
END_VAR
VAR
	pstSysInfo: POINTER TO T_DL_SysInfo;
END_VAR
// methode check, if data log allready exists and if not allocate a new system
// -> return reference on new system

// exist at least one data log system
IF (stDatLogLibInfo.pstDatLogSysInfo=TC3_MEMMAN.NULL) THEN
	// create  a new system
	stDatLogLibInfo.pstDatLogSysInfo := M_AllocMEM(SIZEOF(T_DL_SysInfo));

	IF (stDatLogLibInfo.pstDatLogSysInfo=TC3_MEMMAN.NULL) THEN
		M_CheckAndAppendDatLogInfo := TC3_MEMMAN.NULL;
		RETURN;
	END_IF
	
	// data log name entry in info system
	stDatLogLibInfo.pstDatLogSysInfo^.strDatLogName := In_strDatLogName;
	M_CheckAndAppendDatLogInfo := stDatLogLibInfo.pstDatLogSysInfo;
	RETURN;
END_IF

// after this point the system has to exist
IF (stDatLogLibInfo.pstDatLogSysInfo<>TC3_MEMMAN.NULL) THEN
	pstSysInfo := stDatLogLibInfo.pstDatLogSysInfo;
	
	WHILE (pstSysInfo<>TC3_MEMMAN.NULL) DO
		IF (pstSysInfo^.strDatLogName=In_strDatLogName) THEN
			// data log name found -> return handle
			M_CheckAndAppendDatLogInfo := pstSysInfo;
			RETURN;
		END_IF
		
		// last element
		IF (pstSysInfo^.pstNextDatLogSystem=TC3_MEMMAN.NULL) THEN
			// the requested log name does not exist -> allocate a new one
			pstSysInfo^.pstNextDatLogSystem := M_AllocMEM(SIZEOF(T_DL_SysInfo));

			IF (pstSysInfo^.pstNextDatLogSystem<>TC3_MEMMAN.NULL) THEN
				pstSysInfo := pstSysInfo^.pstNextDatLogSystem;
				// data log name entry in info system
				pstSysInfo^.strDatLogName := In_strDatLogName;
				M_CheckAndAppendDatLogInfo := pstSysInfo;
				RETURN;
			ELSE
				M_CheckAndAppendDatLogInfo := TC3_MEMMAN.NULL;
				RETURN;
			END_IF
		ELSE
			// reference next
			pstSysInfo := pstSysInfo^.pstNextDatLogSystem;
		END_IF
	END_WHILE
END_IF
END_METHOD

METHOD PUBLIC M_GetHandle : UINT
VAR_INPUT
	In_strDatLogName: STRING(DatLog.cMAX_SYS_NAME_LENGTH); // name of the client
	In_p_fbBasLog: POINTER TO FB_BasLog; // only one central FB_BasLog instance allowed per PLC!!!
END_VAR
VAR_OUTPUT
	Out_pHandle : POINTER TO BYTE; // handle of log system for write (M_Log)
	Out_udiStatus : UDINT; //0 => successful done, <>0 => error
END_VAR
VAR
	pstSysInfo: POINTER TO T_DL_SysInfo;
	uinGetHandleStatus : UINT;
END_VAR

// check if log system allready exists or not, if not allocate a new one
	pstSysInfo := M_CheckAndAppendDatLogInfo(In_strDatLogName:=In_strDatLogName);
	IF (pstSysInfo=TC3_MEMMAN.NULL) THEN
		Out_udiStatus := DatLog.cERR_MEM_ALLOC;
		RETURN;
	END_IF
	
	// log on base log system
	uinGetHandleStatus := In_p_fbBasLog^.M_GetHandle(Out_pHandle=>pstSysInfo^.pBaseLogHandle);
	
	// check error
	IF (uinGetHandleStatus<>0) THEN
		Out_udiStatus := UINT_TO_UDINT(uinGetHandleStatus);
		RETURN;
	ELSE
		pstSysInfo^.p_fbBasLog := In_p_fbBasLog;
		Out_pHandle := pstSysInfo;
	END_IF
END_METHOD

METHOD PUBLIC M_Init : BOOL
VAR_INPUT
	In_bolExecute : BOOL;
	In_strDatLogName: STRING(DatLog.cMAX_SYS_NAME_LENGTH); // name of the client
	In_a_strDataDefinition: ARRAY[0..DatLog.cMAX_NR_OF_VAR] OF STRING(DatLog.cMAX_VAR_NAME_LEN); // complete VarName: p.e.:MAIN.INIT_TASK.VARINT
	In_uinStartId: UINT;	// Start ident for item index -> cfg file config has to match with this number!
	In_Port : T_AmsPort;	// on plc the first runtime system is the 801, 811 ...
END_VAR
VAR_OUTPUT
	Out_udiStatus: UDINT;		 // 0 => successful done, <>0 => error
	Out_bolDone: BOOL;			// Done
END_VAR
VAR
	pstSysInfo: POINTER TO T_DL_SysInfo;
	pstItem : POINTER TO T_DL_Item;
	ii : UINT;
END_VAR

IF (In_bolExecute=TRUE) THEN
	// check if log system allready exists or not, if not allocate a new one
	pstSysInfo := M_CheckAndAppendDatLogInfo(In_strDatLogName:=In_strDatLogName);
	IF (pstSysInfo=TC3_MEMMAN.NULL) THEN
		Out_udiStatus := DatLog.cERR_MEM_ALLOC;
		RETURN;
	END_IF

	IF (stDatLogLibInfo.stStatemachine.bolExecute_old=FALSE) THEN // reset statemachine
		stDatLogLibInfo.stStatemachine.uinState := 1;
		Out_bolDone := FALSE;
		Out_udiStatus := 0;
		stDatLogLibInfo.stStatemachine.usiInitDone := 0;
	END_IF

CASE stDatLogLibInfo.stStatemachine.uinState OF
	1:
		//check number of elements
		FOR ii :=0 TO DatLog.cMAX_NR_OF_VAR BY 1 DO
			IF (In_a_strDataDefinition[ii]='') THEN
				EXIT;
			END_IF
		END_FOR
		
		pstSysInfo^.uinNbrOfItems := ii;
		pstSysInfo^.uinStartId := In_uinStartId;
		
		// allocate memory for items
		pstSysInfo^.pstItems := M_AllocMEM((pstSysInfo^.uinNbrOfItems*SIZEOF(T_DL_Item)));
		IF (pstSysInfo^.pstItems =TC3_MEMMAN.NULL) THEN
			Out_udiStatus := DatLog.cERR_MEM_ALLOC;
			RETURN;
		END_IF
		pstSysInfo^.uinCntReadItems := 0;
		pstSysInfo^.uinItemOffset := 0;
		stDatLogLibInfo.stStatemachine.uinState := stDatLogLibInfo.stStatemachine.uinState + 1;
		
	2:	
		fbPLC_ReadSymInfo.NETID:=''; // local PLC
		IF (In_Port=0) THEN// access first runtime system
			fbPLC_ReadSymInfo.PORT := 851;
		ELSE
			fbPLC_ReadSymInfo.PORT := In_Port;
		END_IF
		fbPLC_ReadSymInfo.SYMNAME := In_a_strDataDefinition[pstSysInfo^.uinCntReadItems];
		fbPLC_ReadSymInfo.START := FALSE;
		fbPLC_ReadSymInfo();
		fbPLC_ReadSymInfo.START := TRUE;
		fbPLC_ReadSymInfo();
		stDatLogLibInfo.stStatemachine.uinState := stDatLogLibInfo.stStatemachine.uinState + 1;
		
	3:
		fbPLC_ReadSymInfo();
		IF (fbPLC_ReadSymInfo.BUSY=FALSE) THEN
			stDatLogLibInfo.stStatemachine.uinState := stDatLogLibInfo.stStatemachine.uinState + 1;
		END_IF
		
	4:
		pstItem := pstSysInfo^.pstItems;
		IF (fbPLC_ReadSymInfo.ERR=FALSE) THEN
			pstItem[pstSysInfo^.uinCntReadItems].strPvName := In_a_strDataDefinition[pstSysInfo^.uinCntReadItems];
			pstItem[pstSysInfo^.uinCntReadItems].uinItemOffset := pstSysInfo^.uinItemOffset;
			pstItem[pstSysInfo^.uinCntReadItems].SymInfo := fbPLC_ReadSymInfo.SYMINFO;
			pstSysInfo^.uinItemOffset := pstSysInfo^.uinItemOffset + UDINT_TO_UINT(pstItem[pstSysInfo^.uinCntReadItems].SymInfo.byteSize); // offset for next
			
			// check if type ok/allowed
			IF (pstItem[pstSysInfo^.uinCntReadItems].SymInfo.symDataType = 'BOOL') THEN 
				pstItem[pstSysInfo^.uinCntReadItems].udiItemType := DatLog.cVAR_TYPE_BOOL;
			ELSIF (pstItem[pstSysInfo^.uinCntReadItems].SymInfo.symDataType = 'SINT') THEN 
				pstItem[pstSysInfo^.uinCntReadItems].udiItemType := DatLog.cVAR_TYPE_SINT;
			ELSIF (pstItem[pstSysInfo^.uinCntReadItems].SymInfo.symDataType = 'INT') THEN 
				pstItem[pstSysInfo^.uinCntReadItems].udiItemType := DatLog.cVAR_TYPE_INT;
			ELSIF (pstItem[pstSysInfo^.uinCntReadItems].SymInfo.symDataType = 'DINT') THEN 
				pstItem[pstSysInfo^.uinCntReadItems].udiItemType := DatLog.cVAR_TYPE_DINT;
			ELSIF (pstItem[pstSysInfo^.uinCntReadItems].SymInfo.symDataType = 'USINT') THEN 
				pstItem[pstSysInfo^.uinCntReadItems].udiItemType := DatLog.cVAR_TYPE_USINT;
			ELSIF (pstItem[pstSysInfo^.uinCntReadItems].SymInfo.symDataType = 'UINT') THEN 
				pstItem[pstSysInfo^.uinCntReadItems].udiItemType := DatLog.cVAR_TYPE_INT;
			ELSIF (pstItem[pstSysInfo^.uinCntReadItems].SymInfo.symDataType = 'UDINT') THEN 
				pstItem[pstSysInfo^.uinCntReadItems].udiItemType := DatLog.cVAR_TYPE_UDINT;
			ELSIF (pstItem[pstSysInfo^.uinCntReadItems].SymInfo.symDataType = 'REAL') THEN 
				pstItem[pstSysInfo^.uinCntReadItems].udiItemType := DatLog.cVAR_TYPE_REAL;
			ELSIF (FIND(STR1:=pstItem[pstSysInfo^.uinCntReadItems].SymInfo.symDataType,STR2:='STRING')<>0) THEN 
				IF (pstItem[pstSysInfo^.uinCntReadItems].SymInfo.byteSize < BasLog.cMAX_CHAR_TEXT2) THEN
					pstItem[pstSysInfo^.uinCntReadItems].udiItemType := DatLog.cVAR_TYPE_STRING;
				ELSE
					Out_udiStatus := DatLog.cERR_UNSUPPORTED_TYPE_STRING_TOO_LONG;
					RETURN;
				END_IF
			ELSE
				Out_udiStatus := DatLog.cERR_UNSUPPORTED_TYPE;
				RETURN;
			END_IF
		ELSE
			Out_udiStatus := fbPLC_ReadSymInfo.ERRID;
			RETURN;
		END_IF
		
		pstSysInfo^.uinCntReadItems := pstSysInfo^.uinCntReadItems  + 1;
		IF (pstSysInfo^.uinCntReadItems<pstSysInfo^.uinNbrOfItems) THEN // read next value
			stDatLogLibInfo.stStatemachine.uinState := 2;
		ELSE
			stDatLogLibInfo.stStatemachine.uinState := stDatLogLibInfo.stStatemachine.uinState + 1; // all items found
		END_IF
	5:
		Out_bolDone := TRUE;
		Out_udiStatus := 0;
		pstSysInfo^.usiInitOk := 1; 
END_CASE
END_IF
stDatLogLibInfo.stStatemachine.bolExecute_old := In_bolExecute;
END_METHOD

METHOD PUBLIC M_Log : UINT
VAR_INPUT
	In_pHandle : POINTER TO BYTE;// handle of log system for write (M_Log)
	In_a_pData: ARRAY [0..DatLog.cMAX_NR_OF_VAR] OF POINTER TO BYTE;// address of structure elements
END_VAR
VAR_OUTPUT
	Out_udiStatus: UDINT;		// 0 => successful done, <>0 => error
END_VAR
VAR
	pstSysInfo: POINTER TO T_DL_SysInfo;
	pstItem : POINTER TO T_DL_Item;
	pstItemEle : T_DL_Item;
	ii : UINT;
	strText2: STRING(BasLog.cMAX_CHAR_TEXT2); // informationtext2
	dinPar2 : DINT;
	dinId : DINT;
	uinStatus : UINT;
END_VAR
// check handle ok
IF (In_pHandle=TC3_MEMMAN.NULL) THEN
	M_Log := DatLog.cERR_NO_HANDLE;
	RETURN;
END_IF

// check data
IF (In_a_pData[0]=TC3_MEMMAN.NULL) THEN
	M_Log := DatLog.cERR_NO_DATE;
	RETURN;
END_IF

// access data loggger system info
pstSysInfo := In_pHandle;

// check if init ok
IF (pstSysInfo^.usiInitOk=0) THEN
	M_Log := DatLog.cERR_INIT_FAILED;
	RETURN;
END_IF

// check if items
IF (pstSysInfo^.pstItems=TC3_MEMMAN.NULL) OR (pstSysInfo^.uinNbrOfItems<=0) THEN
	M_Log := DatLog.cERR_NO_ITEMS;
	RETURN;
END_IF
// access item definitions
pstItem := pstSysInfo^.pstItems;

// inc. record id: important the id is inc bevor and after writing of data -> to be sure that no second write is done (MUTEX)
stDatLogLibInfo.udiCommonRecIdx := stDatLogLibInfo.udiCommonRecIdx + 1;
IF (stDatLogLibInfo.udiCommonRecIdx=0) THEN
	stDatLogLibInfo.udiCommonRecIdx := stDatLogLibInfo.udiCommonRecIdx + 1;
END_IF
// write record start
// AE_BL_VAR_TYPE_CMD_NEW_REC
uinStatus := pstSysInfo^.p_fbBasLog^.M_Log(In_pHandle := pstSysInfo^.pBaseLogHandle,In_udiLogType:=BasLog.cLOGTYPE_DATA,In_intCtrlID:=DatLog.cCTRL_ID,In_strText1:='DataLog',In_strText2:='AE_BL_VAR_TYPE_CMD_NEW_REC',In_dinPar1:=0,In_dinPar2:=0,In_dinPar3:=BasLog.cVAR_TYPE_CMD_NEW_REC,In_dinPar4:=UDINT_TO_DINT(stDatLogLibInfo.udiCommonRecIdx));
IF (uinStatus<>0) THEN
	M_Log := uinStatus;
	RETURN;
END_IF

// loop over all items and write data to logger
FOR ii :=0 TO (pstSysInfo^.uinNbrOfItems-1) BY 1 DO
	// write item
	pstItemEle := pstItem[ii]; // for debugging
	// id
	dinId := UINT_TO_DINT(pstSysInfo^.uinStartId + ii);
	IF (pstItem[ii].udiItemType=DatLog.cVAR_TYPE_STRING) THEN
		MEMSET(destAddr:=ADR(strText2),fillByte:=0,n:= SIZEOF(strText2)); // to be sure that a zero is at the end
		// doesn't work with beckhoff...MEMCPY(destAddr := ADR(strText2),srcAddr:= (In_pAdrData + pstItem[ii].uinItemOffset),n:=pstItem[ii].SymInfo.byteSize);
		MEMCPY(destAddr := ADR(strText2),srcAddr:= In_a_pData[ii],n:=pstItem[ii].SymInfo.byteSize);
		dinPar2 := 0;
	ELSE
		strText2 := pstItem[ii].strPvName; // just for info
		MEMCPY(destAddr := ADR(dinPar2),srcAddr:= In_a_pData[ii],n:=pstItem[ii].SymInfo.byteSize);
	END_IF
	
	// log item
	uinStatus := pstSysInfo^.p_fbBasLog^.M_Log(In_pHandle := pstSysInfo^.pBaseLogHandle,In_udiLogType:=BasLog.cLOGTYPE_DATA,In_intCtrlID:=DatLog.cCTRL_ID,In_strText1:='DataLog',In_strText2:=strText2,In_dinPar1:=dinId,In_dinPar2:=dinPar2,In_dinPar3:=UDINT_TO_DINT(pstItem[ii].udiItemType),In_dinPar4:=UDINT_TO_DINT(stDatLogLibInfo.udiCommonRecIdx));

	IF (uinStatus<>0) THEN // no stop write error number
		M_Log := uinStatus;
	END_IF
END_FOR

// write record stop
// AE_BL_VAR_TYPE_CMD_NEW_REC
uinStatus := pstSysInfo^.p_fbBasLog^.M_Log(In_pHandle := pstSysInfo^.pBaseLogHandle,In_udiLogType:=BasLog.cLOGTYPE_DATA,In_intCtrlID:=DatLog.cCTRL_ID,In_strText1:='DataLog',In_strText2:='AE_BL_VAR_TYPE_CMD_END_REC',In_dinPar1:=0,In_dinPar2:=0,In_dinPar3:=BasLog.cVAR_TYPE_CMD_END_REC,In_dinPar4:=UDINT_TO_DINT(stDatLogLibInfo.udiCommonRecIdx));
IF (uinStatus<>0) THEN
	M_Log := uinStatus;
	RETURN;
END_IF

// increment id a second time
stDatLogLibInfo.udiCommonRecIdx := stDatLogLibInfo.udiCommonRecIdx + 1;
IF (stDatLogLibInfo.udiCommonRecIdx=0) THEN
	stDatLogLibInfo.udiCommonRecIdx := stDatLogLibInfo.udiCommonRecIdx + 1;
END_IF
END_METHOD

END_FUNCTION_BLOCK

// POUs/Utility/Logger/DatLog/FB_DatLogTest_Sender
FUNCTION_BLOCK FB_DatLogTest_Sender
VAR_INPUT
	In_p_fbBasLog: POINTER TO FB_BasLog; // only one central FB_BasLog instance allowed per PLC!!!
	In_a_pData: ARRAY [0..DatLog.cMAX_NR_OF_VAR] OF POINTER TO BYTE;
	In_strTaskName: STRING(20);
	In_strValueNameOfData: STRING(20);
END_VAR
VAR_OUTPUT
	Out_bolInit : BOOL := FALSE;
END_VAR
VAR
	bolDone : BOOL;
	pDL_Handle: POINTER TO T_DL_SysInfo;
	udiStatusInit :UDINT;
	udiStatus : UDINT;
	fbDatLog: FB_DatLog;
	a_strDataDefinition :ARRAY[0..DatLog.cMAX_NR_OF_VAR] OF STRING(DatLog.cMAX_VAR_NAME_LEN);
	uinDoLogData : UINT;
	strTemp: T_MaxString;
	strTemp2: T_MaxString;
	ii : UINT;
END_VAR

(*__________________________________________________________________________________________________
¦	
¦	Vistaprint Schweiz GmbH
¦	CH - 8401 Winterthur
¦
¦	www.vistaprint.ch - info@vistaprint.ch
¦___________________________________________________________________________________________________

Function desription:
Example and test programm for testing the data logger system - write data to data log

History:
Version		Date			Author		Comment
---------------------------------------------------------------------------------------------------
0.00.1		02.09.2014		AVME/KVO	Start history
___________________________________________________________________________________________________*)

// system init onetime after start up
IF (Out_bolInit=FALSE) THEN
	
	// TODO :parse a struct on PLC...
	FOR ii := 0 TO DatLog.cMAX_NR_OF_VAR DO
		strTemp := In_strTaskName;
		strTemp := CONCAT(STR1 := strTemp,'.');
		strTemp := CONCAT(STR1 := strTemp,In_strValueNameOfData);
		strTemp := CONCAT(STR1 := strTemp,'.');
		// fillup variable elements of struct, order is important!!!!!!!!!!!!!!!!!!!!
		CASE ii OF
			0:
				strTemp2 := 'bolOk';
			1:
				strTemp2 := 'intCnt';
			2:
				strTemp2 := 'strNewText';
		ELSE
			EXIT;
		END_CASE
		a_strDataDefinition[ii] := CONCAT(STR1 := strTemp,STR2:=strTemp2);
	END_FOR
	
	fbDatLog.M_Init(In_bolExecute := TRUE,In_strDatLogName:= 'DatLog',In_a_strDataDefinition:=a_strDataDefinition,In_Port:=851,In_uinStartId:=100,Out_udiStatus=>udiStatusInit,Out_bolDone=>bolDone);
	IF (bolDone OR (udiStatusInit<>0)) THEN
		fbDatLog.M_Init(In_bolExecute := FALSE,In_strDatLogName:= 'DatLog',In_a_strDataDefinition:=a_strDataDefinition,In_Port:=851,In_uinStartId:=100); // reset statemachine
	
		IF (udiStatusInit=0) THEN
			udiStatusInit := fbDatLog.M_GetHandle(In_strDatLogName:='DatLog',In_p_fbBasLog:=In_p_fbBasLog,Out_pHandle=>pDL_Handle,Out_udiStatus=>udiStatusInit);
		END_IF
		
		Out_bolInit := TRUE;
	END_IF

ELSE
	fbDatLog.M_Init(In_bolExecute := FALSE,In_strDatLogName:= 'DatLog',In_a_strDataDefinition:=a_strDataDefinition,In_Port:=851,In_uinStartId:=100); // reset statemachine
	
END_IF

// write entry data 
IF ((pDL_Handle<>TC3_MEMMAN.NULL) AND (udiStatusInit=0) AND (Out_bolInit=TRUE)) THEN
	fbDatLog.M_Log(In_pHandle:=pDL_Handle,In_a_pData:= In_a_pData,Out_udiStatus=>udiStatus);
END_IF

END_FUNCTION_BLOCK

// POUs/Utility/Logger/FileLc/FB_FileLc
FUNCTION_BLOCK FB_FileLc
VAR_INPUT
END_VAR
VAR_OUTPUT
END_VAR
VAR
	stFileLogClientLibInfo : T_FileLc_LibInfo;
	strInfo: Tc2_System.T_MaxString;	// additional debug Info
	bolExecute_old : BOOL;
END_VAR

(*__________________________________________________________________________________________________
¦	
¦	Vistaprint Schweiz GmbH
¦	CH - 8401 Winterthur
¦
¦	www.vistaprint.ch - info@vistaprint.ch
¦___________________________________________________________________________________________________

Function desription:
File client read out informations from BaseLog system and writes based on a config file the log entries to a file.

History:
Version		Date			Author		Comment
---------------------------------------------------------------------------------------------------
0.00.1		18.08.2014		AVME/KVO	Start history
___________________________________________________________________________________________________*)

